LIN {X 0,Y 517.137,Z 472.821,A -85,B 0,C 180,E1 -4939.23,E2 -4939.23} C_VEL
LIN {X 0,Y 516.862,Z 480.781,A -85,B 0,C 180,E1 -4940.412,E2 -4940.412} C_VEL
LIN {X 0,Y 516.641,Z 488.412,A -85,B 0,C 180,E1 -4941.788,E2 -4941.788} C_VEL
LIN {X 0,Y 516.456,Z 493.749,A -85,B 0,C 180,E1 -4942.965,E2 -4942.965} C_VEL
LIN {X 0,Y 516.387,Z 499.361,A -85,B 0,C 180,E1 -4944.533,E2 -4944.533} C_VEL
LIN {X 0,Y 516.343,Z 503.442,A -85,B 0,C 180,E1 -4946.098,E2 -4946.098} C_VEL
LIN {X 0,Y 516.26,Z 506.121,A -85,B 0,C 180,E1 -4947.659,E2 -4947.659} C_VEL
LIN {X 0,Y 516.156,Z 507.471,A -85,B 0,C 180,E1 -4949.22,E2 -4949.22} C_VEL
LIN {X 0,Y 516.157,Z 507.515,A -85,B 0,C 180,E1 -4950.78,E2 -4950.78} C_VEL
LIN {X 0,Y 516.26,Z 506.249,A -85,B 0,C 180,E1 -4952.341,E2 -4952.341} C_VEL
LIN {X 0,Y 516.343,Z 503.644,A -85,B 0,C 180,E1 -4953.902,E2 -4953.902} C_VEL
LIN {X 0,Y 516.381,Z 499.634,A -85,B 0,C 180,E1 -4955.467,E2 -4955.467} C_VEL
LIN {X 0,Y 516.456,Z 494.108,A -85,B 0,C 180,E1 -4957.035,E2 -4957.035} C_VEL
LIN {X 0,Y 516.597,Z 488.866,A -85,B 0,C 180,E1 -4958.213,E2 -4958.213} C_VEL
LIN {X 0,Y 516.842,Z 481.33,A -85,B 0,C 180,E1 -4959.589,E2 -4959.589} C_VEL
LIN {X 0,Y 517.102,Z 473.48,A -85,B 0,C 180,E1 -4960.771,E2 -4960.771} C_VEL
LIN {X 0,Y 517.53,Z 463.302,A -85,B 0,C 180,E1 -4962.032,E2 -4962.032} C_VEL
LIN {X 0,Y 517.893,Z 452.448,A -85,B 0,C 180,E1 -4963.139,E2 -4963.139} C_VEL
LIN {X 0,Y 518.34,Z 440.597,A -85,B 0,C 180,E1 -4964.126,E2 -4964.126} C_VEL
LIN {X 0,Y 518.79,Z 428.907,A -85,B 0,C 180,E1 -4964.916,E2 -4964.916} C_VEL
LIN {X 0,Y 519.149,Z 416.098,A -85,B 0,C 180,E1 -4965.608,E2 -4965.608} C_VEL
LIN {X 0,Y 519.522,Z 402.223,A -85,B 0,C 180,E1 -4966.176,E2 -4966.176} C_VEL
LIN {X 0,Y 519.479,Z 390.943,A -85,B 0,C 180,E1 -4966.522,E2 -4966.522} C_VEL
LIN {X 0,Y 516.431,Z 377.936,A -85,B 0,C 180,E1 -4966.911,E2 -4966.911} C_VEL
LIN {X 0,Y 516.522,Z 371.712,A -85,B 0,C 180,E1 -4970.142,E2 -4970.142} C_VEL
LIN {X 0,Y 516.595,Z 365.792,A -85,B 0,C 180,E1 -4973.237,E2 -4973.237} C_VEL
LIN {X 0,Y 516.693,Z 360.394,A -85,B 0,C 180,E1 -4976.139,E2 -4976.139} C_VEL
LIN {X 0,Y 516.775,Z 356.239,A -85,B 0,C 180,E1 -4978.424,E2 -4978.424} C_VEL
LIN {X 0,Y 516.89,Z 351.438,A -85,B 0,C 180,E1 -4981.11,E2 -4981.11} C_VEL
LIN {X 0,Y 517.015,Z 346.413,A -85,B 0,C 180,E1 -4983.983,E2 -4983.983} C_VEL
LIN {X 0,Y 517.158,Z 341.688,A -85,B 0,C 180,E1 -4986.723,E2 -4986.723} C_VEL
LIN {X 0,Y 517.069,Z 337.486,A -85,B 0,C 180,E1 -4989.218,E2 -4989.218} C_VEL
LIN {X 0,Y 516.936,Z 336.726,A -85,B 0,C 180,E1 -4989.717,E2 -4989.717} C_VEL
LIN {X 0,Y 516.888,Z 336.727,A -85,B 0,C 180,E1 -4992.831,E2 -4992.831} C_VEL
LIN {X 0,Y 516.928,Z 336.721,A -85,B 0,C 180,E1 -4995.01,E2 -4995.01} C_VEL
LIN {X 0,Y 516.918,Z 336.721,A -85,B 0,C 180,E1 -4998.399,E2 -4998.399} C_VEL
LIN {X 0,Y 516.886,Z 336.725,A -85,B 0,C 180,E1 -5001.284,E2 -5001.284} C_VEL
LIN {X 0,Y 516.876,Z 336.724,A -85,B 0,C 180,E1 -5004.22,E2 -5004.22} C_VEL
LIN {X 0,Y 516.9,Z 336.722,A -85,B 0,C 180,E1 -5007.053,E2 -5007.053} C_VEL
LIN {X 0,Y 516.898,Z 336.726,A -85,B 0,C 180,E1 -5009.796,E2 -5009.796} C_VEL
LIN {X 0,Y 516.932,Z 336.717,A -85,B 0,C 180,E1 -5012.467,E2 -5012.467} C_VEL
LIN {X 0,Y 516.915,Z 336.724,A -85,B 0,C 180,E1 -5015.072,E2 -5015.072} C_VEL
LIN {X 0,Y 516.892,Z 336.725,A -85,B 0,C 180,E1 -5018.462,E2 -5018.462} C_VEL
LIN {X 0,Y 516.906,Z 336.72,A -85,B 0,C 180,E1 -5020.955,E2 -5020.955} C_VEL
LIN {X 0,Y 516.916,Z 336.724,A -85,B 0,C 180,E1 -5023.41,E2 -5023.41} C_VEL
LIN {X 0,Y 516.9,Z 336.72,A -85,B 0,C 180,E1 -5025.834,E2 -5025.834} C_VEL
LIN {X 0,Y 516.972,Z 336.715,A -85,B 0,C 180,E1 -5028.234,E2 -5028.234} C_VEL
LIN {X 0,Y 516.969,Z 336.713,A -85,B 0,C 180,E1 -5031.4,E2 -5031.4} C_VEL
LIN {X 0,Y 517.016,Z 336.708,A -85,B 0,C 180,E1 -5033.757,E2 -5033.757} C_VEL
LIN {X 0,Y 517.087,Z 336.696,A -85,B 0,C 180,E1 -5037.663,E2 -5037.663} C_VEL
LIN {X 0,Y 517.1,Z 336.695,A -85,B 0,C 180,E1 -5040.779,E2 -5040.779} C_VEL
LIN {X 0,Y 517.017,Z 336.708,A -85,B 0,C 180,E1 -5043.117,E2 -5043.117} C_VEL
LIN {X 0,Y 517.009,Z 336.708,A -85,B 0,C 180,E1 -5046.243,E2 -5046.243} C_VEL
LIN {X 0,Y 516.948,Z 336.715,A -85,B 0,C 180,E1 -5049.389,E2 -5049.389} C_VEL
LIN {X 0,Y 516.99,Z 336.714,A -85,B 0,C 180,E1 -5051.824,E2 -5051.824} C_VEL
LIN {X 0,Y 516.951,Z 336.72,A -85,B 0,C 180,E1 -5055.146,E2 -5055.146} C_VEL
LIN {X 0,Y 516.93,Z 336.72,A -85,B 0,C 180,E1 -5058.222,E2 -5058.222} C_VEL
LIN {X 0,Y 516.918,Z 336.722,A -85,B 0,C 180,E1 -5060.701,E2 -5060.701} C_VEL
LIN {X 0,Y 516.917,Z 336.721,A -85,B 0,C 180,E1 -5064.072,E2 -5064.072} C_VEL
LIN {X 0,Y 516.93,Z 336.72,A -85,B 0,C 180,E1 -5066.657,E2 -5066.657} C_VEL
LIN {X 0,Y 516.916,Z 336.718,A -85,B 0,C 180,E1 -5069.523,E2 -5069.523} C_VEL
LIN {X 0,Y 516.9,Z 336.724,A -85,B 0,C 180,E1 -5072.543,E2 -5072.543} C_VEL
LIN {X 0,Y 516.887,Z 336.729,A -85,B 0,C 180,E1 -5075.332,E2 -5075.332} C_VEL
LIN {X 0,Y 516.885,Z 336.724,A -85,B 0,C 180,E1 -5077.943,E2 -5077.943} C_VEL
LIN {X 0,Y 516.887,Z 336.725,A -85,B 0,C 180,E1 -5080.741,E2 -5080.741} C_VEL
LIN {X 0,Y 516.886,Z 336.726,A -85,B 0,C 180,E1 -5082.831,E2 -5082.831} C_VEL
LIN {X 0,Y 516.885,Z 336.726,A -85,B 0,C 180,E1 -5086.097,E2 -5086.097} C_VEL
LIN {X 0,Y 516.92,Z 336.722,A -85,B 0,C 180,E1 -5088.398,E2 -5088.398} C_VEL
LIN {X 0,Y 516.919,Z 336.861,A -85,B 0,C 180,E1 -5091.437,E2 -5091.437} C_VEL
LIN {X 0,Y 518.231,Z 343.552,A -85,B 0,C 180,E1 -5093.848,E2 -5093.848} C_VEL
LIN {X 0,Y 518.639,Z 347.942,A -85,B 0,C 180,E1 -5095.31,E2 -5095.31} C_VEL
LIN {X 0,Y 518.251,Z 357.992,A -85,B 0,C 180,E1 -5098.43,E2 -5098.43} C_VEL
LIN {X 0,Y 517.815,Z 368.768,A -85,B 0,C 180,E1 -5101.638,E2 -5101.638} C_VEL
LIN {X 0,Y 517.515,Z 379.281,A -85,B 0,C 180,E1 -5104.673,E2 -5104.673} C_VEL
LIN {X 0,Y 517.245,Z 389.787,A -85,B 0,C 180,E1 -5107.638,E2 -5107.638} C_VEL
LIN {X 0,Y 517.019,Z 399.95,A -85,B 0,C 180,E1 -5110.437,E2 -5110.437} C_VEL
LIN {X 0,Y 520.612,Z 416.224,A -85,B 0,C 180,E1 -5110.856,E2 -5110.856} C_VEL
LIN {X 0,Y 520.274,Z 431.577,A -85,B 0,C 180,E1 -5111.28,E2 -5111.28} C_VEL
LIN {X 0,Y 519.839,Z 447.124,A -85,B 0,C 180,E1 -5111.883,E2 -5111.883} C_VEL
LIN {X 0,Y 519.381,Z 460.906,A -85,B 0,C 180,E1 -5112.579,E2 -5112.579} C_VEL
LIN {X 0,Y 518.872,Z 475.109,A -85,B 0,C 180,E1 -5113.474,E2 -5113.474} C_VEL
LIN {X 0,Y 518.428,Z 487.049,A -85,B 0,C 180,E1 -5114.389,E2 -5114.389} C_VEL
LIN {X 0,Y 517.9,Z 498.835,A -85,B 0,C 180,E1 -5115.46,E2 -5115.46} C_VEL
LIN {X 0,Y 517.518,Z 509.845,A -85,B 0,C 180,E1 -5116.652,E2 -5116.652} C_VEL
LIN {X 0,Y 517.154,Z 519.174,A -85,B 0,C 180,E1 -5117.84,E2 -5117.84} C_VEL
LIN {X 0,Y 516.913,Z 528.292,A -85,B 0,C 180,E1 -5119.225,E2 -5119.225} C_VEL
LIN {X 0,Y 516.637,Z 535.748,A -85,B 0,C 180,E1 -5120.605,E2 -5120.605} C_VEL
LIN {X 0,Y 516.463,Z 542.699,A -85,B 0,C 180,E1 -5122.179,E2 -5122.179} C_VEL
LIN {X 0,Y 516.36,Z 548.161,A -85,B 0,C 180,E1 -5123.749,E2 -5123.749} C_VEL
LIN {X 0,Y 516.238,Z 552.29,A -85,B 0,C 180,E1 -5125.315,E2 -5125.315} C_VEL
LIN {X 0,Y 516.272,Z 555.183,A -85,B 0,C 180,E1 -5126.878,E2 -5126.878} C_VEL
LIN {X 0,Y 516.189,Z 556.909,A -85,B 0,C 180,E1 -5128.44,E2 -5128.44} C_VEL
LIN {X 0,Y 516.151,Z 557.5,A -85,B 0,C 180,E1 -5130,E2 -5130} C_VEL
LIN {X 0,Y 516.189,Z 556.906,A -85,B 0,C 180,E1 -5131.56,E2 -5131.56} C_VEL
LIN {X 0,Y 516.272,Z 555.179,A -85,B 0,C 180,E1 -5133.121,E2 -5133.121} C_VEL
LIN {X 0,Y 516.238,Z 552.288,A -85,B 0,C 180,E1 -5134.685,E2 -5134.685} C_VEL
LIN {X 0,Y 516.376,Z 548.165,A -85,B 0,C 180,E1 -5136.251,E2 -5136.251} C_VEL
LIN {X 0,Y 516.463,Z 542.7,A -85,B 0,C 180,E1 -5137.821,E2 -5137.821} C_VEL
LIN {X 0,Y 516.637,Z 535.742,A -85,B 0,C 180,E1 -5139.395,E2 -5139.395} C_VEL
LIN {X 0,Y 516.91,Z 528.289,A -85,B 0,C 180,E1 -5140.775,E2 -5140.775} C_VEL
LIN {X 0,Y 517.137,Z 519.449,A -85,B 0,C 180,E1 -5142.121,E2 -5142.121} C_VEL
LIN {X 0,Y 517.518,Z 509.847,A -85,B 0,C 180,E1 -5143.348,E2 -5143.348} C_VEL
LIN {X 0,Y 517.882,Z 498.84,A -85,B 0,C 180,E1 -5144.54,E2 -5144.54} C_VEL
LIN {X 0,Y 518.403,Z 487.055,A -85,B 0,C 180,E1 -5145.612,E2 -5145.612} C_VEL
LIN {X 0,Y 518.922,Z 473.663,A -85,B 0,C 180,E1 -5146.625,E2 -5146.625} C_VEL
LIN {X 0,Y 519.373,Z 460.888,A -85,B 0,C 180,E1 -5147.421,E2 -5147.421} C_VEL
LIN {X 0,Y 519.858,Z 447.119,A -85,B 0,C 180,E1 -5148.116,E2 -5148.116} C_VEL
LIN {X 0,Y 520.27,Z 432.263,A -85,B 0,C 180,E1 -5148.697,E2 -5148.697} C_VEL
LIN {X 0,Y 520.606,Z 416.99,A -85,B 0,C 180,E1 -5149.127,E2 -5149.127} C_VEL
LIN {X 0,Y 519.173,Z 409.765,A -85,B 0,C 180,E1 -5149.329,E2 -5149.329} C_VEL
LIN {X 0,Y 517.014,Z 399.848,A -85,B 0,C 180,E1 -5149.591,E2 -5149.591} C_VEL
LIN {X 0,Y 517.303,Z 388.214,A -85,B 0,C 180,E1 -5152.799,E2 -5152.799} C_VEL
LIN {X 0,Y 517.574,Z 376.755,A -85,B 0,C 180,E1 -5156.05,E2 -5156.05} C_VEL
LIN {X 0,Y 517.876,Z 367.26,A -85,B 0,C 180,E1 -5158.801,E2 -5158.801} C_VEL
LIN {X 0,Y 518.305,Z 356.796,A -85,B 0,C 180,E1 -5161.926,E2 -5161.926} C_VEL
LIN {X 0,Y 518.669,Z 347.929,A -85,B 0,C 180,E1 -5164.688,E2 -5164.688} C_VEL
LIN {X 0,Y 518.204,Z 343.555,A -85,B 0,C 180,E1 -5166.154,E2 -5166.154} C_VEL
LIN {X 0,Y 516.897,Z 336.728,A -85,B 0,C 180,E1 -5168.615,E2 -5168.615} C_VEL
LIN {X 0,Y 516.917,Z 336.72,A -85,B 0,C 180,E1 -5171.775,E2 -5171.775} C_VEL
LIN {X 0,Y 516.896,Z 336.724,A -85,B 0,C 180,E1 -5175.007,E2 -5175.007} C_VEL
LIN {X 0,Y 516.925,Z 336.715,A -85,B 0,C 180,E1 -5178.398,E2 -5178.398} C_VEL
LIN {X 0,Y 516.909,Z 336.726,A -85,B 0,C 180,E1 -5181.287,E2 -5181.287} C_VEL
LIN {X 0,Y 516.894,Z 336.725,A -85,B 0,C 180,E1 -5184.222,E2 -5184.222} C_VEL
LIN {X 0,Y 516.898,Z 336.723,A -85,B 0,C 180,E1 -5187.053,E2 -5187.053} C_VEL
LIN {X 0,Y 516.895,Z 336.726,A -85,B 0,C 180,E1 -5189.797,E2 -5189.797} C_VEL
LIN {X 0,Y 516.93,Z 336.718,A -85,B 0,C 180,E1 -5192.468,E2 -5192.468} C_VEL
LIN {X 0,Y 516.915,Z 336.721,A -85,B 0,C 180,E1 -5195.072,E2 -5195.072} C_VEL
LIN {X 0,Y 516.874,Z 336.726,A -85,B 0,C 180,E1 -5197.622,E2 -5197.622} C_VEL
LIN {X 0,Y 516.936,Z 336.718,A -85,B 0,C 180,E1 -5200.13,E2 -5200.13} C_VEL
LIN {X 0,Y 516.926,Z 336.718,A -85,B 0,C 180,E1 -5202.596,E2 -5202.596} C_VEL
LIN {X 0,Y 516.947,Z 336.718,A -85,B 0,C 180,E1 -5205.03,E2 -5205.03} C_VEL
LIN {X 0,Y 517.01,Z 336.712,A -85,B 0,C 180,E1 -5208.235,E2 -5208.235} C_VEL
LIN {X 0,Y 516.961,Z 336.717,A -85,B 0,C 180,E1 -5211.4,E2 -5211.4} C_VEL
LIN {X 0,Y 517.015,Z 336.705,A -85,B 0,C 180,E1 -5213.757,E2 -5213.757} C_VEL
LIN {X 0,Y 517.088,Z 336.696,A -85,B 0,C 180,E1 -5217.663,E2 -5217.663} C_VEL
LIN {X 0,Y 517.098,Z 336.693,A -85,B 0,C 180,E1 -5220.779,E2 -5220.779} C_VEL
LIN {X 0,Y 517.017,Z 336.711,A -85,B 0,C 180,E1 -5223.117,E2 -5223.117} C_VEL
LIN {X 0,Y 517.015,Z 336.708,A -85,B 0,C 180,E1 -5226.243,E2 -5226.243} C_VEL
LIN {X 0,Y 516.948,Z 336.715,A -85,B 0,C 180,E1 -5229.389,E2 -5229.389} C_VEL
LIN {X 0,Y 516.989,Z 336.714,A -85,B 0,C 180,E1 -5231.824,E2 -5231.824} C_VEL
LIN {X 0,Y 516.95,Z 336.719,A -85,B 0,C 180,E1 -5235.147,E2 -5235.147} C_VEL
LIN {X 0,Y 516.93,Z 336.72,A -85,B 0,C 180,E1 -5238.222,E2 -5238.222} C_VEL
LIN {X 0,Y 516.917,Z 336.718,A -85,B 0,C 180,E1 -5240.701,E2 -5240.701} C_VEL
LIN {X 0,Y 516.917,Z 336.717,A -85,B 0,C 180,E1 -5244.072,E2 -5244.072} C_VEL
LIN {X 0,Y 516.929,Z 336.722,A -85,B 0,C 180,E1 -5246.658,E2 -5246.658} C_VEL
LIN {X 0,Y 516.916,Z 336.718,A -85,B 0,C 180,E1 -5249.524,E2 -5249.524} C_VEL
LIN {X 0,Y 516.9,Z 336.721,A -85,B 0,C 180,E1 -5252.543,E2 -5252.543} C_VEL
LIN {X 0,Y 516.87,Z 336.729,A -85,B 0,C 180,E1 -5255.33,E2 -5255.33} C_VEL
LIN {X 0,Y 516.884,Z 336.723,A -85,B 0,C 180,E1 -5257.943,E2 -5257.943} C_VEL
LIN {X 0,Y 516.886,Z 336.724,A -85,B 0,C 180,E1 -5260.742,E2 -5260.742} C_VEL
LIN {X 0,Y 516.887,Z 336.723,A -85,B 0,C 180,E1 -5262.831,E2 -5262.831} C_VEL
LIN {X 0,Y 516.927,Z 336.722,A -85,B 0,C 180,E1 -5265.01,E2 -5265.01} C_VEL
LIN {X 0,Y 516.919,Z 336.723,A -85,B 0,C 180,E1 -5268.398,E2 -5268.398} C_VEL
LIN {X 0,Y 516.928,Z 336.723,A -85,B 0,C 180,E1 -5270.301,E2 -5270.301} C_VEL
LIN {X 0,Y 516.613,Z 337.308,A -85,B 0,C 180,E1 -5270.735,E2 -5270.735} C_VEL
LIN {X 0,Y 514.727,Z 338.994,A -85,B 0,C 180,E1 -5271.571,E2 -5271.571} C_VEL
LIN {X 0,Y 511.152,Z 341.674,A -85,B 0,C 180,E1 -5272.806,E2 -5272.806} C_VEL
LIN {X 0,Y 510.164,Z 342.833,A -85,B 0,C 180,E1 -5273.448,E2 -5273.448} C_VEL
LIN {X 0,Y 510.094,Z 343.201,A -85,B 0,C 180,E1 -5273.666,E2 -5273.666} C_VEL
LIN {X 0,Y 509.938,Z 348.134,A -85,B 0,C 180,E1 -5276.545,E2 -5276.545} C_VEL
LIN {X 0,Y 509.824,Z 352.985,A -85,B 0,C 180,E1 -5279.333,E2 -5279.333} C_VEL
LIN {X 0,Y 509.759,Z 357.776,A -85,B 0,C 180,E1 -5282.046,E2 -5282.046} C_VEL
LIN {X 0,Y 509.606,Z 362.537,A -85,B 0,C 180,E1 -5284.689,E2 -5284.689} C_VEL
LIN {X 0,Y 509.536,Z 367.804,A -85,B 0,C 180,E1 -5287.537,E2 -5287.537} C_VEL
LIN {X 0,Y 509.391,Z 373.764,A -85,B 0,C 180,E1 -5290.663,E2 -5290.663} C_VEL
LIN {X 0,Y 509.412,Z 378.216,A -85,B 0,C 180,E1 -5292.926,E2 -5292.926} C_VEL
LIN {X 0,Y 512.717,Z 392.09,A -85,B 0,C 180,E1 -5293.347,E2 -5293.347} C_VEL
LIN {X 0,Y 512.896,Z 396.194,A -85,B 0,C 180,E1 -5293.467,E2 -5293.467} C_VEL
LIN {X 0,Y 512.642,Z 409.242,A -85,B 0,C 180,E1 -5293.93,E2 -5293.93} C_VEL
LIN {X 0,Y 512.206,Z 422.905,A -85,B 0,C 180,E1 -5294.583,E2 -5294.583} C_VEL
LIN {X 0,Y 511.681,Z 435.853,A -85,B 0,C 180,E1 -5295.381,E2 -5295.381} C_VEL
LIN {X 0,Y 511.265,Z 447.552,A -85,B 0,C 180,E1 -5296.283,E2 -5296.283} C_VEL
LIN {X 0,Y 510.771,Z 458.23,A -85,B 0,C 180,E1 -5297.282,E2 -5297.282} C_VEL
LIN {X 0,Y 510.383,Z 468.772,A -85,B 0,C 180,E1 -5298.483,E2 -5298.483} C_VEL
LIN {X 0,Y 509.953,Z 477.477,A -85,B 0,C 180,E1 -5299.679,E2 -5299.679} C_VEL
LIN {X 0,Y 509.687,Z 485.805,A -85,B 0,C 180,E1 -5301.076,E2 -5301.076} C_VEL
LIN {X 0,Y 509.438,Z 492.525,A -85,B 0,C 180,E1 -5302.469,E2 -5302.469} C_VEL
LIN {X 0,Y 509.365,Z 498.532,A -85,B 0,C 180,E1 -5304.06,E2 -5304.06} C_VEL
LIN {X 0,Y 509.192,Z 501.971,A -85,B 0,C 180,E1 -5305.25,E2 -5305.25} C_VEL
LIN {X 0,Y 509.269,Z 503.813,A -85,B 0,C 180,E1 -5306.043,E2 -5306.043} C_VEL
LIN {X 0,Y 509.189,Z 506.475,A -85,B 0,C 180,E1 -5307.627,E2 -5307.627} C_VEL
LIN {X 0,Y 509.07,Z 507.818,A -85,B 0,C 180,E1 -5309.209,E2 -5309.209} C_VEL
LIN {X 0,Y 509.071,Z 507.86,A -85,B 0,C 180,E1 -5310.791,E2 -5310.791} C_VEL
LIN {X 0,Y 509.188,Z 506.602,A -85,B 0,C 180,E1 -5312.373,E2 -5312.373} C_VEL
LIN {X 0,Y 509.269,Z 504.011,A -85,B 0,C 180,E1 -5313.957,E2 -5313.957} C_VEL
LIN {X 0,Y 509.318,Z 500.02,A -85,B 0,C 180,E1 -5315.543,E2 -5315.543} C_VEL
LIN {X 0,Y 509.419,Z 494.516,A -85,B 0,C 180,E1 -5317.133,E2 -5317.133} C_VEL
LIN {X 0,Y 509.578,Z 489.301,A -85,B 0,C 180,E1 -5318.327,E2 -5318.327} C_VEL
LIN {X 0,Y 509.847,Z 481.794,A -85,B 0,C 180,E1 -5319.722,E2 -5319.722} C_VEL
LIN {X 0,Y 510.155,Z 473.976,A -85,B 0,C 180,E1 -5320.919,E2 -5320.919} C_VEL
LIN {X 0,Y 510.595,Z 464.033,A -85,B 0,C 180,E1 -5322.175,E2 -5322.175} C_VEL
LIN {X 0,Y 510.998,Z 453.021,A -85,B 0,C 180,E1 -5323.319,E2 -5323.319} C_VEL
LIN {X 0,Y 511.491,Z 441.213,A -85,B 0,C 180,E1 -5324.319,E2 -5324.319} C_VEL
LIN {X 0,Y 511.978,Z 429.575,A -85,B 0,C 180,E1 -5325.119,E2 -5325.119} C_VEL
LIN {X 0,Y 512.36,Z 416.84,A -85,B 0,C 180,E1 -5325.821,E2 -5325.821} C_VEL
LIN {X 0,Y 512.762,Z 403.636,A -85,B 0,C 180,E1 -5326.376,E2 -5326.376} C_VEL
LIN {X 0,Y 512.838,Z 392.563,A -85,B 0,C 180,E1 -5326.726,E2 -5326.726} C_VEL
LIN {X 0,Y 509.841,Z 380.168,A -85,B 0,C 180,E1 -5327.115,E2 -5327.115} C_VEL
LIN {X 0,Y 509.379,Z 378.113,A -85,B 0,C 180,E1 -5327.179,E2 -5327.179} C_VEL
LIN {X 0,Y 509.466,Z 372.16,A -85,B 0,C 180,E1 -5330.273,E2 -5330.273} C_VEL
LIN {X 0,Y 509.517,Z 367.488,A -85,B 0,C 180,E1 -5332.72,E2 -5332.72} C_VEL
LIN {X 0,Y 509.604,Z 362.713,A -85,B 0,C 180,E1 -5335.311,E2 -5335.311} C_VEL
LIN {X 0,Y 509.709,Z 357.756,A -85,B 0,C 180,E1 -5338.06,E2 -5338.06} C_VEL
LIN {X 0,Y 509.852,Z 352.06,A -85,B 0,C 180,E1 -5341.281,E2 -5341.281} C_VEL
LIN {X 0,Y 509.979,Z 346.663,A -85,B 0,C 180,E1 -5344.404,E2 -5344.404} C_VEL
LIN {X 0,Y 510.118,Z 341.73,A -85,B 0,C 180,E1 -5347.316,E2 -5347.316} C_VEL
LIN {X 0,Y 509.957,Z 337.852,A -85,B 0,C 180,E1 -5349.66,E2 -5349.66} C_VEL
LIN {X 0,Y 509.844,Z 337.608,A -85,B 0,C 180,E1 -5350.382,E2 -5350.382} C_VEL
LIN {X 0,Y 509.829,Z 337.607,A -85,B 0,C 180,E1 -5353.062,E2 -5353.062} C_VEL
LIN {X 0,Y 509.835,Z 337.601,A -85,B 0,C 180,E1 -5355.793,E2 -5355.793} C_VEL
LIN {X 0,Y 509.86,Z 337.598,A -85,B 0,C 180,E1 -5358.575,E2 -5358.575} C_VEL
LIN {X 0,Y 509.856,Z 337.601,A -85,B 0,C 180,E1 -5361.787,E2 -5361.787} C_VEL
LIN {X 0,Y 509.835,Z 337.604,A -85,B 0,C 180,E1 -5364.622,E2 -5364.622} C_VEL
LIN {X 0,Y 509.867,Z 337.597,A -85,B 0,C 180,E1 -5367.481,E2 -5367.481} C_VEL
LIN {X 0,Y 509.864,Z 337.6,A -85,B 0,C 180,E1 -5370.274,E2 -5370.274} C_VEL
LIN {X 0,Y 509.889,Z 337.597,A -85,B 0,C 180,E1 -5372.944,E2 -5372.944} C_VEL
LIN {X 0,Y 509.871,Z 337.597,A -85,B 0,C 180,E1 -5375.574,E2 -5375.574} C_VEL
LIN {X 0,Y 509.856,Z 337.596,A -85,B 0,C 180,E1 -5378.998,E2 -5378.998} C_VEL
LIN {X 0,Y 509.867,Z 337.601,A -85,B 0,C 180,E1 -5381.516,E2 -5381.516} C_VEL
LIN {X 0,Y 509.86,Z 337.598,A -85,B 0,C 180,E1 -5383.997,E2 -5383.997} C_VEL
LIN {X 0,Y 509.867,Z 337.599,A -85,B 0,C 180,E1 -5386.448,E2 -5386.448} C_VEL
LIN {X 0,Y 509.92,Z 337.591,A -85,B 0,C 180,E1 -5388.875,E2 -5388.875} C_VEL
LIN {X 0,Y 509.956,Z 337.588,A -85,B 0,C 180,E1 -5392.078,E2 -5392.078} C_VEL
LIN {X 0,Y 509.988,Z 337.581,A -85,B 0,C 180,E1 -5394.464,E2 -5394.464} C_VEL
LIN {X 0,Y 510.059,Z 337.572,A -85,B 0,C 180,E1 -5397.631,E2 -5397.631} C_VEL
LIN {X 0,Y 510.07,Z 337.571,A -85,B 0,C 180,E1 -5400.789,E2 -5400.789} C_VEL
LIN {X 0,Y 509.959,Z 337.587,A -85,B 0,C 180,E1 -5403.16,E2 -5403.16} C_VEL
LIN {X 0,Y 509.96,Z 337.586,A -85,B 0,C 180,E1 -5406.33,E2 -5406.33} C_VEL
LIN {X 0,Y 509.91,Z 337.596,A -85,B 0,C 180,E1 -5408.72,E2 -5408.72} C_VEL
LIN {X 0,Y 509.958,Z 337.591,A -85,B 0,C 180,E1 -5411.93,E2 -5411.93} C_VEL
LIN {X 0,Y 509.9,Z 337.599,A -85,B 0,C 180,E1 -5415.241,E2 -5415.241} C_VEL
LIN {X 0,Y 509.888,Z 337.596,A -85,B 0,C 180,E1 -5417.998,E2 -5417.998} C_VEL
LIN {X 0,Y 509.856,Z 337.6,A -85,B 0,C 180,E1 -5421.001,E2 -5421.001} C_VEL
LIN {X 0,Y 509.842,Z 337.605,A -85,B 0,C 180,E1 -5423.563,E2 -5423.563} C_VEL
LIN {X 0,Y 509.916,Z 337.592,A -85,B 0,C 180,E1 -5426.378,E2 -5426.378} C_VEL
LIN {X 0,Y 509.881,Z 337.6,A -85,B 0,C 180,E1 -5428.844,E2 -5428.844} C_VEL
LIN {X 0,Y 509.824,Z 337.604,A -85,B 0,C 180,E1 -5431.59,E2 -5431.59} C_VEL
LIN {X 0,Y 509.858,Z 337.6,A -85,B 0,C 180,E1 -5434.413,E2 -5434.413} C_VEL
LIN {X 0,Y 509.823,Z 337.607,A -85,B 0,C 180,E1 -5437.34,E2 -5437.34} C_VEL
LIN {X 0,Y 509.841,Z 337.605,A -85,B 0,C 180,E1 -5440.382,E2 -5440.382} C_VEL
LIN {X 0,Y 509.826,Z 337.605,A -85,B 0,C 180,E1 -5443.062,E2 -5443.062} C_VEL
LIN {X 0,Y 509.826,Z 337.608,A -85,B 0,C 180,E1 -5445.793,E2 -5445.793} C_VEL
LIN {X 0,Y 509.861,Z 337.602,A -85,B 0,C 180,E1 -5448.574,E2 -5448.574} C_VEL
LIN {X 0,Y 509.86,Z 337.702,A -85,B 0,C 180,E1 -5451.094,E2 -5451.094} C_VEL
LIN {X 0,Y 511.3,Z 345.012,A -85,B 0,C 180,E1 -5453.768,E2 -5453.768} C_VEL
LIN {X 0,Y 511.7,Z 350.138,A -85,B 0,C 180,E1 -5455.495,E2 -5455.495} C_VEL
LIN {X 0,Y 511.286,Z 359.73,A -85,B 0,C 180,E1 -5458.51,E2 -5458.51} C_VEL
LIN {X 0,Y 510.829,Z 370.314,A -85,B 0,C 180,E1 -5461.704,E2 -5461.704} C_VEL
LIN {X 0,Y 510.494,Z 380.675,A -85,B 0,C 180,E1 -5464.736,E2 -5464.736} C_VEL
LIN {X 0,Y 510.208,Z 391.227,A -85,B 0,C 180,E1 -5467.757,E2 -5467.757} C_VEL
LIN {X 0,Y 509.998,Z 399.799,A -85,B 0,C 180,E1 -5470.178,E2 -5470.178} C_VEL
LIN {X 0,Y 513.494,Z 415.649,A -85,B 0,C 180,E1 -5470.596,E2 -5470.596} C_VEL
LIN {X 0,Y 513.832,Z 419.248,A -85,B 0,C 180,E1 -5470.692,E2 -5470.692} C_VEL
LIN {X 0,Y 513.386,Z 435.11,A -85,B 0,C 180,E1 -5471.177,E2 -5471.177} C_VEL
LIN {X 0,Y 512.942,Z 449.643,A -85,B 0,C 180,E1 -5471.786,E2 -5471.786} C_VEL
LIN {X 0,Y 512.385,Z 463.703,A -85,B 0,C 180,E1 -5472.54,E2 -5472.54} C_VEL
LIN {X 0,Y 511.869,Z 477.307,A -85,B 0,C 180,E1 -5473.447,E2 -5473.447} C_VEL
LIN {X 0,Y 511.349,Z 490.45,A -85,B 0,C 180,E1 -5474.515,E2 -5474.515} C_VEL
LIN {X 0,Y 510.771,Z 502.22,A -85,B 0,C 180,E1 -5475.66,E2 -5475.66} C_VEL
LIN {X 0,Y 510.39,Z 512.629,A -85,B 0,C 180,E1 -5476.867,E2 -5476.867} C_VEL
LIN {X 0,Y 509.935,Z 522.67,A -85,B 0,C 180,E1 -5478.25,E2 -5478.25} C_VEL
LIN {X 0,Y 509.716,Z 531.261,A -85,B 0,C 180,E1 -5479.674,E2 -5479.674} C_VEL
LIN {X 0,Y 509.484,Z 539.186,A -85,B 0,C 180,E1 -5481.272,E2 -5481.272} C_VEL
LIN {X 0,Y 509.318,Z 545.482,A -85,B 0,C 180,E1 -5482.866,E2 -5482.866} C_VEL
LIN {X 0,Y 509.284,Z 550.35,A -85,B 0,C 180,E1 -5484.457,E2 -5484.457} C_VEL
LIN {X 0,Y 509.2,Z 553.885,A -85,B 0,C 180,E1 -5486.043,E2 -5486.043} C_VEL
LIN {X 0,Y 509.158,Z 556.188,A -85,B 0,C 180,E1 -5487.627,E2 -5487.627} C_VEL
LIN {X 0,Y 509.071,Z 557.347,A -85,B 0,C 180,E1 -5489.209,E2 -5489.209} C_VEL
LIN {X 0,Y 509.071,Z 557.346,A -85,B 0,C 180,E1 -5490.791,E2 -5490.791} C_VEL
LIN {X 0,Y 509.158,Z 556.184,A -85,B 0,C 180,E1 -5492.373,E2 -5492.373} C_VEL
LIN {X 0,Y 509.2,Z 553.88,A -85,B 0,C 180,E1 -5493.957,E2 -5493.957} C_VEL
LIN {X 0,Y 509.285,Z 550.351,A -85,B 0,C 180,E1 -5495.543,E2 -5495.543} C_VEL
LIN {X 0,Y 509.32,Z 545.488,A -85,B 0,C 180,E1 -5497.134,E2 -5497.134} C_VEL
LIN {X 0,Y 509.484,Z 539.185,A -85,B 0,C 180,E1 -5498.728,E2 -5498.728} C_VEL
LIN {X 0,Y 509.716,Z 531.258,A -85,B 0,C 180,E1 -5500.326,E2 -5500.326} C_VEL
LIN {X 0,Y 509.964,Z 522.478,A -85,B 0,C 180,E1 -5501.777,E2 -5501.777} C_VEL
LIN {X 0,Y 510.389,Z 512.631,A -85,B 0,C 180,E1 -5503.132,E2 -5503.132} C_VEL
LIN {X 0,Y 510.757,Z 502.221,A -85,B 0,C 180,E1 -5504.34,E2 -5504.34} C_VEL
LIN {X 0,Y 511.29,Z 490.455,A -85,B 0,C 180,E1 -5505.487,E2 -5505.487} C_VEL
LIN {X 0,Y 511.864,Z 477.314,A -85,B 0,C 180,E1 -5506.553,E2 -5506.553} C_VEL
LIN {X 0,Y 512.408,Z 463.701,A -85,B 0,C 180,E1 -5507.459,E2 -5507.459} C_VEL
LIN {X 0,Y 512.899,Z 449.641,A -85,B 0,C 180,E1 -5508.215,E2 -5508.215} C_VEL
LIN {X 0,Y 513.407,Z 435.094,A -85,B 0,C 180,E1 -5508.824,E2 -5508.824} C_VEL
LIN {X 0,Y 513.806,Z 419.604,A -85,B 0,C 180,E1 -5509.3,E2 -5509.3} C_VEL
LIN {X 0,Y 513.494,Z 415.662,A -85,B 0,C 180,E1 -5509.403,E2 -5509.403} C_VEL
LIN {X 0,Y 510.11,Z 400.69,A -85,B 0,C 180,E1 -5509.804,E2 -5509.804} C_VEL
LIN {X 0,Y 509.99,Z 399.71,A -85,B 0,C 180,E1 -5509.838,E2 -5509.838} C_VEL
LIN {X 0,Y 510.3,Z 388.157,A -85,B 0,C 180,E1 -5513.111,E2 -5513.111} C_VEL
LIN {X 0,Y 510.569,Z 377.68,A -85,B 0,C 180,E1 -5516.135,E2 -5516.135} C_VEL
LIN {X 0,Y 510.941,Z 367.168,A -85,B 0,C 180,E1 -5519.229,E2 -5519.229} C_VEL
LIN {X 0,Y 511.34,Z 358.222,A -85,B 0,C 180,E1 -5521.948,E2 -5521.948} C_VEL
LIN {X 0,Y 511.738,Z 349.158,A -85,B 0,C 180,E1 -5524.816,E2 -5524.816} C_VEL
LIN {X 0,Y 511.064,Z 343.845,A -85,B 0,C 180,E1 -5526.645,E2 -5526.645} C_VEL
LIN {X 0,Y 509.856,Z 337.606,A -85,B 0,C 180,E1 -5528.97,E2 -5528.97} C_VEL
LIN {X 0,Y 509.862,Z 337.599,A -85,B 0,C 180,E1 -5531.898,E2 -5531.898} C_VEL
LIN {X 0,Y 509.84,Z 337.602,A -85,B 0,C 180,E1 -5535.33,E2 -5535.33} C_VEL
LIN {X 0,Y 509.868,Z 337.593,A -85,B 0,C 180,E1 -5538.576,E2 -5538.576} C_VEL
LIN {X 0,Y 509.862,Z 337.601,A -85,B 0,C 180,E1 -5541.663,E2 -5541.663} C_VEL
LIN {X 0,Y 509.85,Z 337.606,A -85,B 0,C 180,E1 -5544.624,E2 -5544.624} C_VEL
LIN {X 0,Y 509.864,Z 337.601,A -85,B 0,C 180,E1 -5547.481,E2 -5547.481} C_VEL
LIN {X 0,Y 509.862,Z 337.599,A -85,B 0,C 180,E1 -5550.274,E2 -5550.274} C_VEL
LIN {X 0,Y 509.887,Z 337.6,A -85,B 0,C 180,E1 -5552.945,E2 -5552.945} C_VEL
LIN {X 0,Y 509.874,Z 337.596,A -85,B 0,C 180,E1 -5555.574,E2 -5555.574} C_VEL
LIN {X 0,Y 509.827,Z 337.605,A -85,B 0,C 180,E1 -5558.149,E2 -5558.149} C_VEL
LIN {X 0,Y 509.867,Z 337.596,A -85,B 0,C 180,E1 -5560.682,E2 -5560.682} C_VEL
LIN {X 0,Y 509.887,Z 337.598,A -85,B 0,C 180,E1 -5563.175,E2 -5563.175} C_VEL
LIN {X 0,Y 509.869,Z 337.596,A -85,B 0,C 180,E1 -5565.634,E2 -5565.634} C_VEL
LIN {X 0,Y 509.927,Z 337.589,A -85,B 0,C 180,E1 -5568.875,E2 -5568.875} C_VEL
LIN {X 0,Y 509.926,Z 337.59,A -85,B 0,C 180,E1 -5572.078,E2 -5572.078} C_VEL
LIN {X 0,Y 509.986,Z 337.582,A -85,B 0,C 180,E1 -5574.464,E2 -5574.464} C_VEL
LIN {X 0,Y 510.059,Z 337.571,A -85,B 0,C 180,E1 -5577.631,E2 -5577.631} C_VEL
LIN {X 0,Y 510.068,Z 337.569,A -85,B 0,C 180,E1 -5580.79,E2 -5580.79} C_VEL
LIN {X 0,Y 509.959,Z 337.591,A -85,B 0,C 180,E1 -5583.16,E2 -5583.16} C_VEL
LIN {X 0,Y 509.983,Z 337.585,A -85,B 0,C 180,E1 -5586.33,E2 -5586.33} C_VEL
LIN {X 0,Y 509.914,Z 337.592,A -85,B 0,C 180,E1 -5588.72,E2 -5588.72} C_VEL
LIN {X 0,Y 509.957,Z 337.588,A -85,B 0,C 180,E1 -5591.931,E2 -5591.931} C_VEL
LIN {X 0,Y 509.899,Z 337.596,A -85,B 0,C 180,E1 -5595.242,E2 -5595.242} C_VEL
LIN {X 0,Y 509.887,Z 337.595,A -85,B 0,C 180,E1 -5597.999,E2 -5597.999} C_VEL
LIN {X 0,Y 509.855,Z 337.597,A -85,B 0,C 180,E1 -5601.002,E2 -5601.002} C_VEL
LIN {X 0,Y 509.875,Z 337.594,A -85,B 0,C 180,E1 -5604.426,E2 -5604.426} C_VEL
LIN {X 0,Y 509.888,Z 337.597,A -85,B 0,C 180,E1 -5607.056,E2 -5607.056} C_VEL
LIN {X 0,Y 509.862,Z 337.598,A -85,B 0,C 180,E1 -5609.751,E2 -5609.751} C_VEL
LIN {X 0,Y 509.877,Z 337.595,A -85,B 0,C 180,E1 -5612.774,E2 -5612.774} C_VEL
LIN {X 0,Y 509.83,Z 337.604,A -85,B 0,C 180,E1 -5615.578,E2 -5615.578} C_VEL
LIN {X 0,Y 509.854,Z 337.602,A -85,B 0,C 180,E1 -5618.338,E2 -5618.338} C_VEL
LIN {X 0,Y 509.859,Z 337.6,A -85,B 0,C 180,E1 -5621.425,E2 -5621.425} C_VEL
LIN {X 0,Y 509.86,Z 337.599,A -85,B 0,C 180,E1 -5624.668,E2 -5624.668} C_VEL
LIN {X 0,Y 509.861,Z 337.601,A -85,B 0,C 180,E1 -5628.103,E2 -5628.103} C_VEL
LIN {X 0,Y 509.9,Z 337.701,A -85,B 0,C 180,E1 -5630.343,E2 -5630.343} C_VEL
LIN {X 0,Y 510.095,Z 341.555,A -85,B 0,C 180,E1 -5632.683,E2 -5632.683} C_VEL
LIN {X 0,Y 510.094,Z 343.201,A -85,B 0,C 180,E1 -5633.666,E2 -5633.666} C_VEL
LIN {X 0,Y 509.45,Z 344.397,A -85,B 0,C 180,E1 -5634.311,E2 -5634.311} C_VEL
LIN {X 0,Y 506.569,Z 346.569,A -85,B 0,C 180,E1 -5635.352,E2 -5635.352} C_VEL
LIN {X 0,Y 504.089,Z 348.346,A -85,B 0,C 180,E1 -5636.19,E2 -5636.19} C_VEL
LIN {X 0,Y 502.985,Z 349.605,A -85,B 0,C 180,E1 -5636.84,E2 -5636.84} C_VEL
LIN {X 0,Y 502.877,Z 349.996,A -85,B 0,C 180,E1 -5637.061,E2 -5637.061} C_VEL
LIN {X 0,Y 502.761,Z 355.185,A -85,B 0,C 180,E1 -5640.076,E2 -5640.076} C_VEL
LIN {X 0,Y 502.681,Z 359.482,A -85,B 0,C 180,E1 -5642.524,E2 -5642.524} C_VEL
LIN {X 0,Y 502.545,Z 364.564,A -85,B 0,C 180,E1 -5645.37,E2 -5645.37} C_VEL
LIN {X 0,Y 502.463,Z 369.048,A -85,B 0,C 180,E1 -5647.812,E2 -5647.812} C_VEL
LIN {X 0,Y 502.339,Z 373.908,A -85,B 0,C 180,E1 -5650.38,E2 -5650.38} C_VEL
LIN {X 0,Y 502.358,Z 378.329,A -85,B 0,C 180,E1 -5652.649,E2 -5652.649} C_VEL
LIN {X 0,Y 505.974,Z 393.158,A -85,B 0,C 180,E1 -5653.118,E2 -5653.118} C_VEL
LIN {X 0,Y 506.134,Z 397.717,A -85,B 0,C 180,E1 -5653.258,E2 -5653.258} C_VEL
LIN {X 0,Y 505.813,Z 411.196,A -85,B 0,C 180,E1 -5653.758,E2 -5653.758} C_VEL
LIN {X 0,Y 505.412,Z 423.631,A -85,B 0,C 180,E1 -5654.37,E2 -5654.37} C_VEL
LIN {X 0,Y 504.863,Z 436.516,A -85,B 0,C 180,E1 -5655.179,E2 -5655.179} C_VEL
LIN {X 0,Y 504.408,Z 448.16,A -85,B 0,C 180,E1 -5656.093,E2 -5656.093} C_VEL
LIN {X 0,Y 503.875,Z 458.794,A -85,B 0,C 180,E1 -5657.105,E2 -5657.105} C_VEL
LIN {X 0,Y 503.444,Z 469.296,A -85,B 0,C 180,E1 -5658.322,E2 -5658.322} C_VEL
LIN {X 0,Y 502.975,Z 477.966,A -85,B 0,C 180,E1 -5659.534,E2 -5659.534} C_VEL
LIN {X 0,Y 502.68,Z 486.261,A -85,B 0,C 180,E1 -5660.951,E2 -5660.951} C_VEL
LIN {X 0,Y 502.418,Z 492.95,A -85,B 0,C 180,E1 -5662.363,E2 -5662.363} C_VEL
LIN {X 0,Y 502.284,Z 497.566,A -85,B 0,C 180,E1 -5663.573,E2 -5663.573} C_VEL
LIN {X 0,Y 502.176,Z 501.307,A -85,B 0,C 180,E1 -5664.781,E2 -5664.781} C_VEL
LIN {X 0,Y 502.198,Z 504.183,A -85,B 0,C 180,E1 -5665.988,E2 -5665.988} C_VEL
LIN {X 0,Y 502.119,Z 506.83,A -85,B 0,C 180,E1 -5667.594,E2 -5667.594} C_VEL
LIN {X 0,Y 501.987,Z 508.164,A -85,B 0,C 180,E1 -5669.198,E2 -5669.198} C_VEL
LIN {X 0,Y 501.988,Z 508.206,A -85,B 0,C 180,E1 -5670.802,E2 -5670.802} C_VEL
LIN {X 0,Y 502.119,Z 506.954,A -85,B 0,C 180,E1 -5672.407,E2 -5672.407} C_VEL
LIN {X 0,Y 502.198,Z 504.379,A -85,B 0,C 180,E1 -5674.013,E2 -5674.013} C_VEL
LIN {X 0,Y 502.258,Z 500.406,A -85,B 0,C 180,E1 -5675.621,E2 -5675.621} C_VEL
LIN {X 0,Y 502.367,Z 494.928,A -85,B 0,C 180,E1 -5677.233,E2 -5677.233} C_VEL
LIN {X 0,Y 502.565,Z 489.736,A -85,B 0,C 180,E1 -5678.444,E2 -5678.444} C_VEL
LIN {X 0,Y 502.852,Z 482.259,A -85,B 0,C 180,E1 -5679.858,E2 -5679.858} C_VEL
LIN {X 0,Y 503.203,Z 474.473,A -85,B 0,C 180,E1 -5681.072,E2 -5681.072} C_VEL
LIN {X 0,Y 503.611,Z 465.494,A -85,B 0,C 180,E1 -5682.239,E2 -5682.239} C_VEL
LIN {X 0,Y 504.1,Z 454.648,A -85,B 0,C 180,E1 -5683.402,E2 -5683.402} C_VEL
LIN {X 0,Y 504.594,Z 443.109,A -85,B 0,C 180,E1 -5684.416,E2 -5684.416} C_VEL
LIN {X 0,Y 505.126,Z 431.818,A -85,B 0,C 180,E1 -5685.225,E2 -5685.225} C_VEL
LIN {X 0,Y 505.485,Z 419.575,A -85,B 0,C 180,E1 -5685.938,E2 -5685.938} C_VEL
LIN {X 0,Y 505.949,Z 405.734,A -85,B 0,C 180,E1 -5686.553,E2 -5686.553} C_VEL
LIN {X 0,Y 506.113,Z 393.977,A -85,B 0,C 180,E1 -5686.944,E2 -5686.944} C_VEL
LIN {X 0,Y 503.36,Z 382.326,A -85,B 0,C 180,E1 -5687.329,E2 -5687.329} C_VEL
LIN {X 0,Y 502.321,Z 378.296,A -85,B 0,C 180,E1 -5687.451,E2 -5687.451} C_VEL
LIN {X 0,Y 502.412,Z 372.472,A -85,B 0,C 180,E1 -5690.47,E2 -5690.47} C_VEL
LIN {X 0,Y 502.467,Z 367.604,A -85,B 0,C 180,E1 -5693.057,E2 -5693.057} C_VEL
LIN {X 0,Y 502.571,Z 362.838,A -85,B 0,C 180,E1 -5695.691,E2 -5695.691} C_VEL
LIN {X 0,Y 502.664,Z 358.061,A -85,B 0,C 180,E1 -5698.384,E2 -5698.384} C_VEL
LIN {X 0,Y 502.799,Z 353.227,A -85,B 0,C 180,E1 -5701.143,E2 -5701.143} C_VEL
LIN {X 0,Y 502.94,Z 348.372,A -85,B 0,C 180,E1 -5703.984,E2 -5703.984} C_VEL
LIN {X 0,Y 503.091,Z 343.436,A -85,B 0,C 180,E1 -5706.92,E2 -5706.92} C_VEL
LIN {X 0,Y 503.055,Z 340.084,A -85,B 0,C 180,E1 -5708.953,E2 -5708.953} C_VEL
LIN {X 0,Y 502.844,Z 338.482,A -85,B 0,C 180,E1 -5710.01,E2 -5710.01} C_VEL
LIN {X 0,Y 502.778,Z 338.485,A -85,B 0,C 180,E1 -5713.231,E2 -5713.231} C_VEL
LIN {X 0,Y 502.794,Z 338.478,A -85,B 0,C 180,E1 -5715.661,E2 -5715.661} C_VEL
LIN {X 0,Y 502.823,Z 338.473,A -85,B 0,C 180,E1 -5719.005,E2 -5719.005} C_VEL
LIN {X 0,Y 502.798,Z 338.478,A -85,B 0,C 180,E1 -5722.046,E2 -5722.046} C_VEL
LIN {X 0,Y 502.804,Z 338.481,A -85,B 0,C 180,E1 -5725.034,E2 -5725.034} C_VEL
LIN {X 0,Y 502.789,Z 338.481,A -85,B 0,C 180,E1 -5727.916,E2 -5727.916} C_VEL
LIN {X 0,Y 502.83,Z 338.474,A -85,B 0,C 180,E1 -5730.712,E2 -5730.712} C_VEL
LIN {X 0,Y 502.868,Z 338.471,A -85,B 0,C 180,E1 -5733.439,E2 -5733.439} C_VEL
LIN {X 0,Y 502.792,Z 338.479,A -85,B 0,C 180,E1 -5736.086,E2 -5736.086} C_VEL
LIN {X 0,Y 502.79,Z 338.478,A -85,B 0,C 180,E1 -5738.689,E2 -5738.689} C_VEL
LIN {X 0,Y 502.832,Z 338.475,A -85,B 0,C 180,E1 -5741.248,E2 -5741.248} C_VEL
LIN {X 0,Y 502.855,Z 338.471,A -85,B 0,C 180,E1 -5744.6,E2 -5744.6} C_VEL
LIN {X 0,Y 502.883,Z 338.468,A -85,B 0,C 180,E1 -5748.039,E2 -5748.039} C_VEL
LIN {X 0,Y 502.874,Z 338.467,A -85,B 0,C 180,E1 -5751.157,E2 -5751.157} C_VEL
LIN {X 0,Y 502.934,Z 338.464,A -85,B 0,C 180,E1 -5753.581,E2 -5753.581} C_VEL
LIN {X 0,Y 502.904,Z 338.47,A -85,B 0,C 180,E1 -5756.795,E2 -5756.795} C_VEL
LIN {X 0,Y 503.04,Z 338.447,A -85,B 0,C 180,E1 -5759.199,E2 -5759.199} C_VEL
LIN {X 0,Y 502.907,Z 338.466,A -85,B 0,C 180,E1 -5761.601,E2 -5761.601} C_VEL
LIN {X 0,Y 502.902,Z 338.467,A -85,B 0,C 180,E1 -5763.204,E2 -5763.204} C_VEL
LIN {X 0,Y 502.913,Z 338.465,A -85,B 0,C 180,E1 -5766.419,E2 -5766.419} C_VEL
LIN {X 0,Y 502.87,Z 338.472,A -85,B 0,C 180,E1 -5768.843,E2 -5768.843} C_VEL
LIN {X 0,Y 502.9,Z 338.47,A -85,B 0,C 180,E1 -5772.1,E2 -5772.1} C_VEL
LIN {X 0,Y 502.854,Z 338.477,A -85,B 0,C 180,E1 -5775.399,E2 -5775.399} C_VEL
LIN {X 0,Y 502.846,Z 338.474,A -85,B 0,C 180,E1 -5778.12,E2 -5778.12} C_VEL
LIN {X 0,Y 502.834,Z 338.478,A -85,B 0,C 180,E1 -5780.536,E2 -5780.536} C_VEL
LIN {X 0,Y 502.803,Z 338.477,A -85,B 0,C 180,E1 -5783.04,E2 -5783.04} C_VEL
LIN {X 0,Y 502.845,Z 338.475,A -85,B 0,C 180,E1 -5785.675,E2 -5785.675} C_VEL
LIN {X 0,Y 502.844,Z 338.474,A -85,B 0,C 180,E1 -5788.372,E2 -5788.372} C_VEL
LIN {X 0,Y 502.797,Z 338.479,A -85,B 0,C 180,E1 -5791.498,E2 -5791.498} C_VEL
LIN {X 0,Y 502.811,Z 338.478,A -85,B 0,C 180,E1 -5794.444,E2 -5794.444} C_VEL
LIN {X 0,Y 502.785,Z 338.485,A -85,B 0,C 180,E1 -5797.178,E2 -5797.178} C_VEL
LIN {X 0,Y 502.791,Z 338.479,A -85,B 0,C 180,E1 -5800.015,E2 -5800.015} C_VEL
LIN {X 0,Y 502.806,Z 338.483,A -85,B 0,C 180,E1 -5802.199,E2 -5802.199} C_VEL
LIN {X 0,Y 502.789,Z 338.483,A -85,B 0,C 180,E1 -5805.47,E2 -5805.47} C_VEL
LIN {X 0,Y 502.833,Z 338.477,A -85,B 0,C 180,E1 -5807.864,E2 -5807.864} C_VEL
LIN {X 0,Y 502.834,Z 338.616,A -85,B 0,C 180,E1 -5810.768,E2 -5810.768} C_VEL
LIN {X 0,Y 504.327,Z 346.191,A -85,B 0,C 180,E1 -5813.589,E2 -5813.589} C_VEL
LIN {X 0,Y 504.804,Z 350.933,A -85,B 0,C 180,E1 -5815.226,E2 -5815.226} C_VEL
LIN {X 0,Y 504.343,Z 360.257,A -85,B 0,C 180,E1 -5818.215,E2 -5818.215} C_VEL
LIN {X 0,Y 503.857,Z 370.921,A -85,B 0,C 180,E1 -5821.492,E2 -5821.492} C_VEL
LIN {X 0,Y 503.505,Z 380.571,A -85,B 0,C 180,E1 -5824.36,E2 -5824.36} C_VEL
LIN {X 0,Y 503.193,Z 391.349,A -85,B 0,C 180,E1 -5827.513,E2 -5827.513} C_VEL
LIN {X 0,Y 502.954,Z 399.565,A -85,B 0,C 180,E1 -5829.906,E2 -5829.906} C_VEL
LIN {X 0,Y 506.604,Z 416.317,A -85,B 0,C 180,E1 -5830.365,E2 -5830.365} C_VEL
LIN {X 0,Y 507.059,Z 419.412,A -85,B 0,C 180,E1 -5830.457,E2 -5830.457} C_VEL
LIN {X 0,Y 506.589,Z 434.07,A -85,B 0,C 180,E1 -5830.908,E2 -5830.908} C_VEL
LIN {X 0,Y 506.143,Z 448.869,A -85,B 0,C 180,E1 -5831.533,E2 -5831.533} C_VEL
LIN {X 0,Y 505.551,Z 463,A -85,B 0,C 180,E1 -5832.296,E2 -5832.296} C_VEL
LIN {X 0,Y 504.976,Z 476.662,A -85,B 0,C 180,E1 -5833.214,E2 -5833.214} C_VEL
LIN {X 0,Y 504.414,Z 489.155,A -85,B 0,C 180,E1 -5834.234,E2 -5834.234} C_VEL
LIN {X 0,Y 503.788,Z 501.667,A -85,B 0,C 180,E1 -5835.457,E2 -5835.457} C_VEL
LIN {X 0,Y 503.369,Z 512.106,A -85,B 0,C 180,E1 -5836.681,E2 -5836.681} C_VEL
LIN {X 0,Y 502.865,Z 521.93,A -85,B 0,C 180,E1 -5838.045,E2 -5838.045} C_VEL
LIN {X 0,Y 502.742,Z 529.671,A -85,B 0,C 180,E1 -5839.325,E2 -5839.325} C_VEL
LIN {X 0,Y 502.449,Z 536.918,A -85,B 0,C 180,E1 -5840.743,E2 -5840.743} C_VEL
LIN {X 0,Y 502.276,Z 543.633,A -85,B 0,C 180,E1 -5842.361,E2 -5842.361} C_VEL
LIN {X 0,Y 502.167,Z 548.358,A -85,B 0,C 180,E1 -5843.784,E2 -5843.784} C_VEL
LIN {X 0,Y 502.081,Z 551.909,A -85,B 0,C 180,E1 -5845.182,E2 -5845.182} C_VEL
LIN {X 0,Y 502.107,Z 554.868,A -85,B 0,C 180,E1 -5846.79,E2 -5846.79} C_VEL
LIN {X 0,Y 502.033,Z 556.626,A -85,B 0,C 180,E1 -5848.396,E2 -5848.396} C_VEL
LIN {X 0,Y 501.977,Z 557.227,A -85,B 0,C 180,E1 -5850,E2 -5850} C_VEL
LIN {X 0,Y 502.033,Z 556.625,A -85,B 0,C 180,E1 -5851.604,E2 -5851.604} C_VEL
LIN {X 0,Y 502.107,Z 554.865,A -85,B 0,C 180,E1 -5853.21,E2 -5853.21} C_VEL
LIN {X 0,Y 502.081,Z 551.911,A -85,B 0,C 180,E1 -5854.818,E2 -5854.818} C_VEL
LIN {X 0,Y 502.233,Z 547.705,A -85,B 0,C 180,E1 -5856.428,E2 -5856.428} C_VEL
LIN {X 0,Y 502.3,Z 542.115,A -85,B 0,C 180,E1 -5858.043,E2 -5858.043} C_VEL
LIN {X 0,Y 502.462,Z 534.997,A -85,B 0,C 180,E1 -5859.663,E2 -5859.663} C_VEL
LIN {X 0,Y 502.797,Z 527.384,A -85,B 0,C 180,E1 -5861.081,E2 -5861.081} C_VEL
LIN {X 0,Y 503.115,Z 518.194,A -85,B 0,C 180,E1 -5862.505,E2 -5862.505} C_VEL
LIN {X 0,Y 503.573,Z 507.115,A -85,B 0,C 180,E1 -5863.931,E2 -5863.931} C_VEL
LIN {X 0,Y 504.086,Z 495.723,A -85,B 0,C 180,E1 -5865.154,E2 -5865.154} C_VEL
LIN {X 0,Y 504.666,Z 483.217,A -85,B 0,C 180,E1 -5866.276,E2 -5866.276} C_VEL
LIN {X 0,Y 505.273,Z 469.402,A -85,B 0,C 180,E1 -5867.296,E2 -5867.296} C_VEL
LIN {X 0,Y 505.822,Z 455.858,A -85,B 0,C 180,E1 -5868.113,E2 -5868.113} C_VEL
LIN {X 0,Y 506.418,Z 441.17,A -85,B 0,C 180,E1 -5868.813,E2 -5868.813} C_VEL
LIN {X 0,Y 506.848,Z 426.364,A -85,B 0,C 180,E1 -5869.349,E2 -5869.349} C_VEL
LIN {X 0,Y 506.846,Z 417.327,A -85,B 0,C 180,E1 -5869.602,E2 -5869.602} C_VEL
LIN {X 0,Y 503.486,Z 402.282,A -85,B 0,C 180,E1 -5870.027,E2 -5870.027} C_VEL
LIN {X 0,Y 502.953,Z 399.509,A -85,B 0,C 180,E1 -5870.11,E2 -5870.11} C_VEL
LIN {X 0,Y 503.301,Z 388.035,A -85,B 0,C 180,E1 -5873.451,E2 -5873.451} C_VEL
LIN {X 0,Y 503.616,Z 377.574,A -85,B 0,C 180,E1 -5876.523,E2 -5876.523} C_VEL
LIN {X 0,Y 504.016,Z 367.077,A -85,B 0,C 180,E1 -5879.671,E2 -5879.671} C_VEL
LIN {X 0,Y 504.407,Z 358.159,A -85,B 0,C 180,E1 -5882.441,E2 -5882.441} C_VEL
LIN {X 0,Y 504.807,Z 350.808,A -85,B 0,C 180,E1 -5884.807,E2 -5884.807} C_VEL
LIN {X 0,Y 504.297,Z 346.182,A -85,B 0,C 180,E1 -5886.41,E2 -5886.41} C_VEL
LIN {X 0,Y 502.807,Z 338.485,A -85,B 0,C 180,E1 -5889.298,E2 -5889.298} C_VEL
LIN {X 0,Y 502.804,Z 338.479,A -85,B 0,C 180,E1 -5892.199,E2 -5892.199} C_VEL
LIN {X 0,Y 502.787,Z 338.481,A -85,B 0,C 180,E1 -5895.47,E2 -5895.47} C_VEL
LIN {X 0,Y 502.829,Z 338.47,A -85,B 0,C 180,E1 -5898.935,E2 -5898.935} C_VEL
LIN {X 0,Y 502.8,Z 338.479,A -85,B 0,C 180,E1 -5902.047,E2 -5902.047} C_VEL
LIN {X 0,Y 502.813,Z 338.48,A -85,B 0,C 180,E1 -5905.035,E2 -5905.035} C_VEL
LIN {X 0,Y 502.786,Z 338.486,A -85,B 0,C 180,E1 -5907.916,E2 -5907.916} C_VEL
LIN {X 0,Y 502.827,Z 338.475,A -85,B 0,C 180,E1 -5910.713,E2 -5910.713} C_VEL
LIN {X 0,Y 502.866,Z 338.471,A -85,B 0,C 180,E1 -5913.44,E2 -5913.44} C_VEL
LIN {X 0,Y 502.796,Z 338.481,A -85,B 0,C 180,E1 -5916.087,E2 -5916.087} C_VEL
LIN {X 0,Y 502.788,Z 338.477,A -85,B 0,C 180,E1 -5918.689,E2 -5918.689} C_VEL
LIN {X 0,Y 502.833,Z 338.477,A -85,B 0,C 180,E1 -5921.249,E2 -5921.249} C_VEL
LIN {X 0,Y 502.826,Z 338.472,A -85,B 0,C 180,E1 -5923.767,E2 -5923.767} C_VEL
LIN {X 0,Y 502.836,Z 338.476,A -85,B 0,C 180,E1 -5926.255,E2 -5926.255} C_VEL
LIN {X 0,Y 502.897,Z 338.466,A -85,B 0,C 180,E1 -5928.717,E2 -5928.717} C_VEL
LIN {X 0,Y 502.885,Z 338.468,A -85,B 0,C 180,E1 -5931.967,E2 -5931.967} C_VEL
LIN {X 0,Y 502.943,Z 338.459,A -85,B 0,C 180,E1 -5934.387,E2 -5934.387} C_VEL
LIN {X 0,Y 503.029,Z 338.447,A -85,B 0,C 180,E1 -5937.598,E2 -5937.598} C_VEL
LIN {X 0,Y 503.033,Z 338.45,A -85,B 0,C 180,E1 -5940,E2 -5940} C_VEL
LIN {X 0,Y 503.028,Z 338.449,A -85,B 0,C 180,E1 -5942.402,E2 -5942.402} C_VEL
LIN {X 0,Y 502.943,Z 338.46,A -85,B 0,C 180,E1 -5945.614,E2 -5945.614} C_VEL
LIN {X 0,Y 502.905,Z 338.465,A -85,B 0,C 180,E1 -5948.033,E2 -5948.033} C_VEL
LIN {X 0,Y 502.898,Z 338.466,A -85,B 0,C 180,E1 -5951.283,E2 -5951.283} C_VEL
LIN {X 0,Y 502.85,Z 338.471,A -85,B 0,C 180,E1 -5954.571,E2 -5954.571} C_VEL
LIN {X 0,Y 502.86,Z 338.47,A -85,B 0,C 180,E1 -5957.907,E2 -5957.907} C_VEL
LIN {X 0,Y 502.834,Z 338.473,A -85,B 0,C 180,E1 -5960.536,E2 -5960.536} C_VEL
LIN {X 0,Y 502.799,Z 338.479,A -85,B 0,C 180,E1 -5963.04,E2 -5963.04} C_VEL
LIN {X 0,Y 502.845,Z 338.472,A -85,B 0,C 180,E1 -5965.675,E2 -5965.675} C_VEL
LIN {X 0,Y 502.844,Z 338.476,A -85,B 0,C 180,E1 -5968.373,E2 -5968.373} C_VEL
LIN {X 0,Y 502.797,Z 338.48,A -85,B 0,C 180,E1 -5971.499,E2 -5971.499} C_VEL
LIN {X 0,Y 502.808,Z 338.478,A -85,B 0,C 180,E1 -5973.994,E2 -5973.994} C_VEL
LIN {X 0,Y 502.781,Z 338.483,A -85,B 0,C 180,E1 -5977.178,E2 -5977.178} C_VEL
LIN {X 0,Y 502.791,Z 338.483,A -85,B 0,C 180,E1 -5980.015,E2 -5980.015} C_VEL
LIN {X 0,Y 502.806,Z 338.48,A -85,B 0,C 180,E1 -5982.199,E2 -5982.199} C_VEL
LIN {X 0,Y 502.805,Z 338.482,A -85,B 0,C 180,E1 -5985.468,E2 -5985.468} C_VEL
LIN {X 0,Y 502.824,Z 338.479,A -85,B 0,C 180,E1 -5988.934,E2 -5988.934} C_VEL
LIN {X 0,Y 502.859,Z 338.647,A -85,B 0,C 180,E1 -5990.236,E2 -5990.236} C_VEL
LIN {X 0,Y 503.073,Z 341.612,A -85,B 0,C 180,E1 -5992.071,E2 -5992.071} C_VEL
LIN {X 0,Y 502.991,Z 346.561,A -85,B 0,C 180,E1 -5995.049,E2 -5995.049} C_VEL
LIN {X 0,Y 502.877,Z 349.996,A -85,B 0,C 180,E1 -5997.061,E2 -5997.061} C_VEL
LIN {X 0,Y 502.156,Z 351.209,A -85,B 0,C 180,E1 -5997.715,E2 -5997.715} C_VEL
LIN {X 0,Y 499.263,Z 353.403,A -85,B 0,C 180,E1 -5998.771,E2 -5998.771} C_VEL
LIN {X 0,Y 496.83,Z 355.175,A -85,B 0,C 180,E1 -5999.622,E2 -5999.622} C_VEL
LIN {X 0,Y 495.766,Z 356.44,A -85,B 0,C 180,E1 -6000.281,E2 -6000.281} C_VEL
LIN {X 0,Y 495.667,Z 356.838,A -85,B 0,C 180,E1 -6000.505,E2 -6000.505} C_VEL
LIN {X 0,Y 495.574,Z 361.716,A -85,B 0,C 180,E1 -6003.309,E2 -6003.309} C_VEL
LIN {X 0,Y 495.468,Z 365.971,A -85,B 0,C 180,E1 -6005.71,E2 -6005.71} C_VEL
LIN {X 0,Y 495.377,Z 370.803,A -85,B 0,C 180,E1 -6008.354,E2 -6008.354} C_VEL
LIN {X 0,Y 495.299,Z 377.584,A -85,B 0,C 180,E1 -6011.933,E2 -6011.933} C_VEL
LIN {X 0,Y 495.326,Z 378.432,A -85,B 0,C 180,E1 -6012.372,E2 -6012.372} C_VEL
LIN {X 0,Y 499.106,Z 393.646,A -85,B 0,C 180,E1 -6012.862,E2 -6012.862} C_VEL
LIN {X 0,Y 499.441,Z 396.933,A -85,B 0,C 180,E1 -6012.968,E2 -6012.968} C_VEL
LIN {X 0,Y 499.125,Z 410.824,A -85,B 0,C 180,E1 -6013.479,E2 -6013.479} C_VEL
LIN {X 0,Y 498.673,Z 422.587,A -85,B 0,C 180,E1 -6014.049,E2 -6014.049} C_VEL
LIN {X 0,Y 498.141,Z 435.772,A -85,B 0,C 180,E1 -6014.87,E2 -6014.87} C_VEL
LIN {X 0,Y 497.583,Z 447.627,A -85,B 0,C 180,E1 -6015.794,E2 -6015.794} C_VEL
LIN {X 0,Y 497.107,Z 457.445,A -85,B 0,C 180,E1 -6016.718,E2 -6016.718} C_VEL
LIN {X 0,Y 496.57,Z 468.227,A -85,B 0,C 180,E1 -6017.95,E2 -6017.95} C_VEL
LIN {X 0,Y 496.116,Z 477.123,A -85,B 0,C 180,E1 -6019.181,E2 -6019.181} C_VEL
LIN {X 0,Y 495.686,Z 485.626,A -85,B 0,C 180,E1 -6020.616,E2 -6020.616} C_VEL
LIN {X 0,Y 495.498,Z 491.606,A -85,B 0,C 180,E1 -6021.846,E2 -6021.846} C_VEL
LIN {X 0,Y 495.252,Z 497.966,A -85,B 0,C 180,E1 -6023.481,E2 -6023.481} C_VEL
LIN {X 0,Y 495.116,Z 501.691,A -85,B 0,C 180,E1 -6024.706,E2 -6024.706} C_VEL
LIN {X 0,Y 495.129,Z 504.552,A -85,B 0,C 180,E1 -6025.93,E2 -6025.93} C_VEL
LIN {X 0,Y 495.052,Z 507.184,A -85,B 0,C 180,E1 -6027.559,E2 -6027.559} C_VEL
LIN {X 0,Y 494.908,Z 508.511,A -85,B 0,C 180,E1 -6029.186,E2 -6029.186} C_VEL
LIN {X 0,Y 494.908,Z 508.551,A -85,B 0,C 180,E1 -6030.814,E2 -6030.814} C_VEL
LIN {X 0,Y 495.052,Z 507.306,A -85,B 0,C 180,E1 -6032.441,E2 -6032.441} C_VEL
LIN {X 0,Y 495.129,Z 504.745,A -85,B 0,C 180,E1 -6034.07,E2 -6034.07} C_VEL
LIN {X 0,Y 495.201,Z 500.792,A -85,B 0,C 180,E1 -6035.702,E2 -6035.702} C_VEL
LIN {X 0,Y 495.318,Z 495.342,A -85,B 0,C 180,E1 -6037.337,E2 -6037.337} C_VEL
LIN {X 0,Y 495.53,Z 490.172,A -85,B 0,C 180,E1 -6038.564,E2 -6038.564} C_VEL
LIN {X 0,Y 495.845,Z 482.728,A -85,B 0,C 180,E1 -6039.999,E2 -6039.999} C_VEL
LIN {X 0,Y 496.256,Z 474.971,A -85,B 0,C 180,E1 -6041.229,E2 -6041.229} C_VEL
LIN {X 0,Y 496.778,Z 464.963,A -85,B 0,C 180,E1 -6042.536,E2 -6042.536} C_VEL
LIN {X 0,Y 497.205,Z 455.237,A -85,B 0,C 180,E1 -6043.592,E2 -6043.592} C_VEL
LIN {X 0,Y 497.761,Z 443.746,A -85,B 0,C 180,E1 -6044.619,E2 -6044.619} C_VEL
LIN {X 0,Y 498.365,Z 430.937,A -85,B 0,C 180,E1 -6045.542,E2 -6045.542} C_VEL
LIN {X 0,Y 498.876,Z 417.33,A -85,B 0,C 180,E1 -6046.313,E2 -6046.313} C_VEL
LIN {X 0,Y 499.283,Z 403.978,A -85,B 0,C 180,E1 -6046.885,E2 -6046.885} C_VEL
LIN {X 0,Y 499.339,Z 395.019,A -85,B 0,C 180,E1 -6047.181,E2 -6047.181} C_VEL
LIN {X 0,Y 496.512,Z 383.182,A -85,B 0,C 180,E1 -6047.587,E2 -6047.587} C_VEL
LIN {X 0,Y 495.277,Z 378.411,A -85,B 0,C 180,E1 -6047.728,E2 -6047.728} C_VEL
LIN {X 0,Y 495.363,Z 372.609,A -85,B 0,C 180,E1 -6050.775,E2 -6050.775} C_VEL
LIN {X 0,Y 495.421,Z 367.742,A -85,B 0,C 180,E1 -6053.404,E2 -6053.404} C_VEL
LIN {X 0,Y 495.522,Z 362.97,A -85,B 0,C 180,E1 -6056.083,E2 -6056.083} C_VEL
LIN {X 0,Y 495.634,Z 358.169,A -85,B 0,C 180,E1 -6058.824,E2 -6058.824} C_VEL
LIN {X 0,Y 495.778,Z 353.162,A -85,B 0,C 180,E1 -6061.729,E2 -6061.729} C_VEL
LIN {X 0,Y 495.928,Z 348.128,A -85,B 0,C 180,E1 -6064.72,E2 -6064.72} C_VEL
LIN {X 0,Y 496.102,Z 343.479,A -85,B 0,C 180,E1 -6067.529,E2 -6067.529} C_VEL
LIN {X 0,Y 495.903,Z 340.112,A -85,B 0,C 180,E1 -6069.624,E2 -6069.624} C_VEL
LIN {X 0,Y 495.791,Z 339.36,A -85,B 0,C 180,E1 -6070.164,E2 -6070.164} C_VEL
LIN {X 0,Y 495.731,Z 339.363,A -85,B 0,C 180,E1 -6072.883,E2 -6072.883} C_VEL
LIN {X 0,Y 495.738,Z 339.358,A -85,B 0,C 180,E1 -6075.999,E2 -6075.999} C_VEL
LIN {X 0,Y 495.771,Z 339.352,A -85,B 0,C 180,E1 -6079.3,E2 -6079.3} C_VEL
LIN {X 0,Y 495.734,Z 339.357,A -85,B 0,C 180,E1 -6082.439,E2 -6082.439} C_VEL
LIN {X 0,Y 495.783,Z 339.352,A -85,B 0,C 180,E1 -6085.457,E2 -6085.457} C_VEL
LIN {X 0,Y 495.761,Z 339.359,A -85,B 0,C 180,E1 -6088.364,E2 -6088.364} C_VEL
LIN {X 0,Y 495.793,Z 339.355,A -85,B 0,C 180,E1 -6091.507,E2 -6091.507} C_VEL
LIN {X 0,Y 495.796,Z 339.349,A -85,B 0,C 180,E1 -6093.932,E2 -6093.932} C_VEL
LIN {X 0,Y 495.766,Z 339.354,A -85,B 0,C 180,E1 -6097.139,E2 -6097.139} C_VEL
LIN {X 0,Y 495.777,Z 339.357,A -85,B 0,C 180,E1 -6100.11,E2 -6100.11} C_VEL
LIN {X 0,Y 495.771,Z 339.352,A -85,B 0,C 180,E1 -6102.681,E2 -6102.681} C_VEL
LIN {X 0,Y 495.796,Z 339.353,A -85,B 0,C 180,E1 -6105.217,E2 -6105.217} C_VEL
LIN {X 0,Y 495.858,Z 339.346,A -85,B 0,C 180,E1 -6108.555,E2 -6108.555} C_VEL
LIN {X 0,Y 495.878,Z 339.343,A -85,B 0,C 180,E1 -6111.852,E2 -6111.852} C_VEL
LIN {X 0,Y 495.902,Z 339.335,A -85,B 0,C 180,E1 -6114.306,E2 -6114.306} C_VEL
LIN {X 0,Y 495.998,Z 339.323,A -85,B 0,C 180,E1 -6117.564,E2 -6117.564} C_VEL
LIN {X 0,Y 495.99,Z 339.325,A -85,B 0,C 180,E1 -6120.812,E2 -6120.812} C_VEL
LIN {X 0,Y 495.999,Z 339.325,A -85,B 0,C 180,E1 -6122.436,E2 -6122.436} C_VEL
LIN {X 0,Y 495.895,Z 339.338,A -85,B 0,C 180,E1 -6125.693,E2 -6125.693} C_VEL
LIN {X 0,Y 495.842,Z 339.344,A -85,B 0,C 180,E1 -6128.148,E2 -6128.148} C_VEL
LIN {X 0,Y 495.879,Z 339.339,A -85,B 0,C 180,E1 -6131.444,E2 -6131.444} C_VEL
LIN {X 0,Y 495.796,Z 339.351,A -85,B 0,C 180,E1 -6134.783,E2 -6134.783} C_VEL
LIN {X 0,Y 495.787,Z 339.354,A -85,B 0,C 180,E1 -6137.318,E2 -6137.318} C_VEL
LIN {X 0,Y 495.776,Z 339.355,A -85,B 0,C 180,E1 -6139.89,E2 -6139.89} C_VEL
LIN {X 0,Y 495.771,Z 339.353,A -85,B 0,C 180,E1 -6142.862,E2 -6142.862} C_VEL
LIN {X 0,Y 495.796,Z 339.35,A -85,B 0,C 180,E1 -6146.067,E2 -6146.067} C_VEL
LIN {X 0,Y 495.777,Z 339.357,A -85,B 0,C 180,E1 -6148.814,E2 -6148.814} C_VEL
LIN {X 0,Y 495.759,Z 339.358,A -85,B 0,C 180,E1 -6151.725,E2 -6151.725} C_VEL
LIN {X 0,Y 495.78,Z 339.353,A -85,B 0,C 180,E1 -6154.695,E2 -6154.695} C_VEL
LIN {X 0,Y 495.735,Z 339.36,A -85,B 0,C 180,E1 -6157.561,E2 -6157.561} C_VEL
LIN {X 0,Y 495.77,Z 339.357,A -85,B 0,C 180,E1 -6160.699,E2 -6160.699} C_VEL
LIN {X 0,Y 495.73,Z 339.362,A -85,B 0,C 180,E1 -6164.001,E2 -6164.001} C_VEL
LIN {X 0,Y 495.76,Z 339.36,A -85,B 0,C 180,E1 -6167.12,E2 -6167.12} C_VEL
LIN {X 0,Y 495.761,Z 339.36,A -85,B 0,C 180,E1 -6169.953,E2 -6169.953} C_VEL
LIN {X 0,Y 495.774,Z 339.498,A -85,B 0,C 180,E1 -6170.419,E2 -6170.419} C_VEL
LIN {X 0,Y 497.162,Z 346.461,A -85,B 0,C 180,E1 -6173.073,E2 -6173.073} C_VEL
LIN {X 0,Y 497.868,Z 351.758,A -85,B 0,C 180,E1 -6174.959,E2 -6174.959} C_VEL
LIN {X 0,Y 497.424,Z 360.951,A -85,B 0,C 180,E1 -6177.965,E2 -6177.965} C_VEL
LIN {X 0,Y 496.911,Z 371.51,A -85,B 0,C 180,E1 -6181.269,E2 -6181.269} C_VEL
LIN {X 0,Y 496.55,Z 380.448,A -85,B 0,C 180,E1 -6183.975,E2 -6183.975} C_VEL
LIN {X 0,Y 496.21,Z 390.639,A -85,B 0,C 180,E1 -6187.016,E2 -6187.016} C_VEL
LIN {X 0,Y 495.925,Z 399.484,A -85,B 0,C 180,E1 -6189.637,E2 -6189.637} C_VEL
LIN {X 0,Y 499.438,Z 415.796,A -85,B 0,C 180,E1 -6190.089,E2 -6190.089} C_VEL
LIN {X 0,Y 500.27,Z 420.477,A -85,B 0,C 180,E1 -6190.242,E2 -6190.242} C_VEL
LIN {X 0,Y 499.785,Z 434.363,A -85,B 0,C 180,E1 -6190.684,E2 -6190.684} C_VEL
LIN {X 0,Y 499.275,Z 449.118,A -85,B 0,C 180,E1 -6191.322,E2 -6191.322} C_VEL
LIN {X 0,Y 498.634,Z 463.917,A -85,B 0,C 180,E1 -6192.148,E2 -6192.148} C_VEL
LIN {X 0,Y 498.016,Z 477.338,A -85,B 0,C 180,E1 -6193.078,E2 -6193.078} C_VEL
LIN {X 0,Y 497.411,Z 490.191,A -85,B 0,C 180,E1 -6194.159,E2 -6194.159} C_VEL
LIN {X 0,Y 496.805,Z 501.102,A -85,B 0,C 180,E1 -6195.248,E2 -6195.248} C_VEL
LIN {X 0,Y 496.357,Z 511.583,A -85,B 0,C 180,E1 -6196.489,E2 -6196.489} C_VEL
LIN {X 0,Y 495.932,Z 520.459,A -85,B 0,C 180,E1 -6197.727,E2 -6197.727} C_VEL
LIN {X 0,Y 495.693,Z 529.217,A -85,B 0,C 180,E1 -6199.172,E2 -6199.172} C_VEL
LIN {X 0,Y 495.361,Z 536.488,A -85,B 0,C 180,E1 -6200.61,E2 -6200.61} C_VEL
LIN {X 0,Y 495.186,Z 543.229,A -85,B 0,C 180,E1 -6202.251,E2 -6202.251} C_VEL
LIN {X 0,Y 495.07,Z 548.305,A -85,B 0,C 180,E1 -6203.815,E2 -6203.815} C_VEL
LIN {X 0,Y 495.006,Z 551.54,A -85,B 0,C 180,E1 -6205.113,E2 -6205.113} C_VEL
LIN {X 0,Y 495.027,Z 554.511,A -85,B 0,C 180,E1 -6206.744,E2 -6206.744} C_VEL
LIN {X 0,Y 494.959,Z 556.279,A -85,B 0,C 180,E1 -6208.373,E2 -6208.373} C_VEL
LIN {X 0,Y 494.895,Z 556.882,A -85,B 0,C 180,E1 -6210,E2 -6210} C_VEL
LIN {X 0,Y 494.959,Z 556.277,A -85,B 0,C 180,E1 -6211.627,E2 -6211.627} C_VEL
LIN {X 0,Y 495.027,Z 554.51,A -85,B 0,C 180,E1 -6213.255,E2 -6213.255} C_VEL
LIN {X 0,Y 495.006,Z 551.544,A -85,B 0,C 180,E1 -6214.887,E2 -6214.887} C_VEL
LIN {X 0,Y 495.161,Z 547.318,A -85,B 0,C 180,E1 -6216.52,E2 -6216.52} C_VEL
LIN {X 0,Y 495.233,Z 541.705,A -85,B 0,C 180,E1 -6218.159,E2 -6218.159} C_VEL
LIN {X 0,Y 495.397,Z 534.559,A -85,B 0,C 180,E1 -6219.802,E2 -6219.802} C_VEL
LIN {X 0,Y 495.733,Z 526.918,A -85,B 0,C 180,E1 -6221.241,E2 -6221.241} C_VEL
LIN {X 0,Y 496.092,Z 517.7,A -85,B 0,C 180,E1 -6222.685,E2 -6222.685} C_VEL
LIN {X 0,Y 496.596,Z 506.574,A -85,B 0,C 180,E1 -6224.13,E2 -6224.13} C_VEL
LIN {X 0,Y 497.113,Z 495.129,A -85,B 0,C 180,E1 -6225.372,E2 -6225.372} C_VEL
LIN {X 0,Y 497.771,Z 482.571,A -85,B 0,C 180,E1 -6226.508,E2 -6226.508} C_VEL
LIN {X 0,Y 498.421,Z 468.692,A -85,B 0,C 180,E1 -6227.542,E2 -6227.542} C_VEL
LIN {X 0,Y 499,Z 455.084,A -85,B 0,C 180,E1 -6228.369,E2 -6228.369} C_VEL
LIN {X 0,Y 499.617,Z 440.713,A -85,B 0,C 180,E1 -6229.062,E2 -6229.062} C_VEL
LIN {X 0,Y 500.079,Z 425.721,A -85,B 0,C 180,E1 -6229.61,E2 -6229.61} C_VEL
LIN {X 0,Y 500.171,Z 418.991,A -85,B 0,C 180,E1 -6229.805,E2 -6229.805} C_VEL
LIN {X 0,Y 496.958,Z 404.323,A -85,B 0,C 180,E1 -6230.243,E2 -6230.243} C_VEL
LIN {X 0,Y 495.921,Z 399.394,A -85,B 0,C 180,E1 -6230.387,E2 -6230.387} C_VEL
LIN {X 0,Y 496.259,Z 389.386,A -85,B 0,C 180,E1 -6233.362,E2 -6233.362} C_VEL
LIN {X 0,Y 496.6,Z 378.954,A -85,B 0,C 180,E1 -6236.474,E2 -6236.474} C_VEL
LIN {X 0,Y 497.047,Z 368.463,A -85,B 0,C 180,E1 -6239.662,E2 -6239.662} C_VEL
LIN {X 0,Y 497.461,Z 359.569,A -85,B 0,C 180,E1 -6242.47,E2 -6242.47} C_VEL
LIN {X 0,Y 497.862,Z 351.73,A -85,B 0,C 180,E1 -6245.04,E2 -6245.04} C_VEL
LIN {X 0,Y 497.398,Z 347.871,A -85,B 0,C 180,E1 -6246.402,E2 -6246.402} C_VEL
LIN {X 0,Y 495.872,Z 339.919,A -85,B 0,C 180,E1 -6249.406,E2 -6249.406} C_VEL
LIN {X 0,Y 495.761,Z 339.363,A -85,B 0,C 180,E1 -6249.638,E2 -6249.638} C_VEL
LIN {X 0,Y 495.739,Z 339.361,A -85,B 0,C 180,E1 -6252.507,E2 -6252.507} C_VEL
LIN {X 0,Y 495.739,Z 339.36,A -85,B 0,C 180,E1 -6255.141,E2 -6255.141} C_VEL
LIN {X 0,Y 495.763,Z 339.352,A -85,B 0,C 180,E1 -6258.22,E2 -6258.22} C_VEL
LIN {X 0,Y 495.781,Z 339.358,A -85,B 0,C 180,E1 -6261.23,E2 -6261.23} C_VEL
LIN {X 0,Y 495.761,Z 339.361,A -85,B 0,C 180,E1 -6264.463,E2 -6264.463} C_VEL
LIN {X 0,Y 495.77,Z 339.356,A -85,B 0,C 180,E1 -6267.406,E2 -6267.406} C_VEL
LIN {X 0,Y 495.769,Z 339.354,A -85,B 0,C 180,E1 -6270.254,E2 -6270.254} C_VEL
LIN {X 0,Y 495.827,Z 339.35,A -85,B 0,C 180,E1 -6273.251,E2 -6273.251} C_VEL
LIN {X 0,Y 495.756,Z 339.355,A -85,B 0,C 180,E1 -6275.725,E2 -6275.725} C_VEL
LIN {X 0,Y 495.748,Z 339.356,A -85,B 0,C 180,E1 -6278.371,E2 -6278.371} C_VEL
LIN {X 0,Y 495.788,Z 339.352,A -85,B 0,C 180,E1 -6280.972,E2 -6280.972} C_VEL
LIN {X 0,Y 495.782,Z 339.351,A -85,B 0,C 180,E1 -6283.53,E2 -6283.53} C_VEL
LIN {X 0,Y 495.799,Z 339.351,A -85,B 0,C 180,E1 -6286.056,E2 -6286.056} C_VEL
LIN {X 0,Y 495.872,Z 339.342,A -85,B 0,C 180,E1 -6288.555,E2 -6288.555} C_VEL
LIN {X 0,Y 495.841,Z 339.346,A -85,B 0,C 180,E1 -6291.852,E2 -6291.852} C_VEL
LIN {X 0,Y 495.9,Z 339.336,A -85,B 0,C 180,E1 -6294.307,E2 -6294.307} C_VEL
LIN {X 0,Y 495.998,Z 339.323,A -85,B 0,C 180,E1 -6297.564,E2 -6297.564} C_VEL
LIN {X 0,Y 496.004,Z 339.325,A -85,B 0,C 180,E1 -6300,E2 -6300} C_VEL
LIN {X 0,Y 495.997,Z 339.325,A -85,B 0,C 180,E1 -6302.436,E2 -6302.436} C_VEL
LIN {X 0,Y 495.901,Z 339.337,A -85,B 0,C 180,E1 -6305.694,E2 -6305.694} C_VEL
LIN {X 0,Y 495.876,Z 339.341,A -85,B 0,C 180,E1 -6308.148,E2 -6308.148} C_VEL
LIN {X 0,Y 495.873,Z 339.342,A -85,B 0,C 180,E1 -6311.445,E2 -6311.445} C_VEL
LIN {X 0,Y 495.795,Z 339.352,A -85,B 0,C 180,E1 -6314.783,E2 -6314.783} C_VEL
LIN {X 0,Y 495.787,Z 339.35,A -85,B 0,C 180,E1 -6317.319,E2 -6317.319} C_VEL
LIN {X 0,Y 495.776,Z 339.356,A -85,B 0,C 180,E1 -6319.89,E2 -6319.89} C_VEL
LIN {X 0,Y 495.766,Z 339.354,A -85,B 0,C 180,E1 -6322.861,E2 -6322.861} C_VEL
LIN {X 0,Y 495.795,Z 339.35,A -85,B 0,C 180,E1 -6326.068,E2 -6326.068} C_VEL
LIN {X 0,Y 495.776,Z 339.353,A -85,B 0,C 180,E1 -6328.815,E2 -6328.815} C_VEL
LIN {X 0,Y 495.76,Z 339.359,A -85,B 0,C 180,E1 -6331.725,E2 -6331.725} C_VEL
LIN {X 0,Y 495.773,Z 339.354,A -85,B 0,C 180,E1 -6334.694,E2 -6334.694} C_VEL
LIN {X 0,Y 495.733,Z 339.358,A -85,B 0,C 180,E1 -6337.562,E2 -6337.562} C_VEL
LIN {X 0,Y 495.77,Z 339.355,A -85,B 0,C 180,E1 -6340.7,E2 -6340.7} C_VEL
LIN {X 0,Y 495.738,Z 339.361,A -85,B 0,C 180,E1 -6344.001,E2 -6344.001} C_VEL
LIN {X 0,Y 495.73,Z 339.364,A -85,B 0,C 180,E1 -6347.117,E2 -6347.117} C_VEL
LIN {X 0,Y 495.816,Z 339.409,A -85,B 0,C 180,E1 -6350.014,E2 -6350.014} C_VEL
LIN {X 0,Y 496.068,Z 343.321,A -85,B 0,C 180,E1 -6352.468,E2 -6352.468} C_VEL
LIN {X 0,Y 495.947,Z 348.283,A -85,B 0,C 180,E1 -6355.47,E2 -6355.47} C_VEL
LIN {X 0,Y 495.779,Z 353.171,A -85,B 0,C 180,E1 -6358.365,E2 -6358.365} C_VEL
LIN {X 0,Y 495.667,Z 356.838,A -85,B 0,C 180,E1 -6360.505,E2 -6360.505} C_VEL
LIN {X 0,Y 494.962,Z 358.08,A -85,B 0,C 180,E1 -6361.168,E2 -6361.168} C_VEL
LIN {X 0,Y 492.07,Z 360.287,A -85,B 0,C 180,E1 -6362.239,E2 -6362.239} C_VEL
LIN {X 0,Y 489.63,Z 362.075,A -85,B 0,C 180,E1 -6363.101,E2 -6363.101} C_VEL
LIN {X 0,Y 488.564,Z 363.362,A -85,B 0,C 180,E1 -6363.77,E2 -6363.77} C_VEL
LIN {X 0,Y 488.467,Z 363.769,A -85,B 0,C 180,E1 -6363.997,E2 -6363.997} C_VEL
LIN {X 0,Y 488.379,Z 367.725,A -85,B 0,C 180,E1 -6366.238,E2 -6366.238} C_VEL
LIN {X 0,Y 488.279,Z 373.345,A -85,B 0,C 180,E1 -6369.321,E2 -6369.321} C_VEL
LIN {X 0,Y 488.237,Z 378.556,A -85,B 0,C 180,E1 -6372.08,E2 -6372.08} C_VEL
LIN {X 0,Y 492.217,Z 394.149,A -85,B 0,C 180,E1 -6372.597,E2 -6372.597} C_VEL
LIN {X 0,Y 492.74,Z 397.327,A -85,B 0,C 180,E1 -6372.71,E2 -6372.71} C_VEL
LIN {X 0,Y 492.427,Z 410.458,A -85,B 0,C 180,E1 -6373.193,E2 -6373.193} C_VEL
LIN {X 0,Y 491.901,Z 423.338,A -85,B 0,C 180,E1 -6373.823,E2 -6373.823} C_VEL
LIN {X 0,Y 491.341,Z 436.451,A -85,B 0,C 180,E1 -6374.656,E2 -6374.656} C_VEL
LIN {X 0,Y 490.726,Z 448.263,A -85,B 0,C 180,E1 -6375.591,E2 -6375.591} C_VEL
LIN {X 0,Y 490.22,Z 458.042,A -85,B 0,C 180,E1 -6376.528,E2 -6376.528} C_VEL
LIN {X 0,Y 489.713,Z 467.181,A -85,B 0,C 180,E1 -6377.569,E2 -6377.569} C_VEL
LIN {X 0,Y 489.255,Z 476.315,A -85,B 0,C 180,E1 -6378.818,E2 -6378.818} C_VEL
LIN {X 0,Y 488.782,Z 485.012,A -85,B 0,C 180,E1 -6380.273,E2 -6380.273} C_VEL
LIN {X 0,Y 488.469,Z 492.048,A -85,B 0,C 180,E1 -6381.728,E2 -6381.728} C_VEL
LIN {X 0,Y 488.202,Z 498.373,A -85,B 0,C 180,E1 -6383.387,E2 -6383.387} C_VEL
LIN {X 0,Y 488.059,Z 502.074,A -85,B 0,C 180,E1 -6384.629,E2 -6384.629} C_VEL
LIN {X 0,Y 488.063,Z 504.921,A -85,B 0,C 180,E1 -6385.871,E2 -6385.871} C_VEL
LIN {X 0,Y 487.987,Z 507.539,A -85,B 0,C 180,E1 -6387.524,E2 -6387.524} C_VEL
LIN {X 0,Y 487.831,Z 508.857,A -85,B 0,C 180,E1 -6389.175,E2 -6389.175} C_VEL
LIN {X 0,Y 487.831,Z 508.896,A -85,B 0,C 180,E1 -6390.826,E2 -6390.826} C_VEL
LIN {X 0,Y 487.987,Z 507.658,A -85,B 0,C 180,E1 -6392.476,E2 -6392.476} C_VEL
LIN {X 0,Y 488.063,Z 505.113,A -85,B 0,C 180,E1 -6394.129,E2 -6394.129} C_VEL
LIN {X 0,Y 488.149,Z 501.184,A -85,B 0,C 180,E1 -6395.784,E2 -6395.784} C_VEL
LIN {X 0,Y 488.295,Z 495.76,A -85,B 0,C 180,E1 -6397.443,E2 -6397.443} C_VEL
LIN {X 0,Y 488.513,Z 490.623,A -85,B 0,C 180,E1 -6398.688,E2 -6398.688} C_VEL
LIN {X 0,Y 488.862,Z 483.217,A -85,B 0,C 180,E1 -6400.143,E2 -6400.143} C_VEL
LIN {X 0,Y 489.315,Z 475.5,A -85,B 0,C 180,E1 -6401.39,E2 -6401.39} C_VEL
LIN {X 0,Y 489.854,Z 465.83,A -85,B 0,C 180,E1 -6402.68,E2 -6402.68} C_VEL
LIN {X 0,Y 490.342,Z 455.841,A -85,B 0,C 180,E1 -6403.785,E2 -6403.785} C_VEL
LIN {X 0,Y 490.941,Z 444.39,A -85,B 0,C 180,E1 -6404.826,E2 -6404.826} C_VEL
LIN {X 0,Y 491.526,Z 433.204,A -85,B 0,C 180,E1 -6405.657,E2 -6405.657} C_VEL
LIN {X 0,Y 491.986,Z 420.088,A -85,B 0,C 180,E1 -6406.441,E2 -6406.441} C_VEL
LIN {X 0,Y 492.52,Z 406.257,A -85,B 0,C 180,E1 -6407.065,E2 -6407.065} C_VEL
LIN {X 0,Y 492.596,Z 396.195,A -85,B 0,C 180,E1 -6407.419,E2 -6407.419} C_VEL
LIN {X 0,Y 489.5,Z 383.517,A -85,B 0,C 180,E1 -6407.867,E2 -6407.867} C_VEL
LIN {X 0,Y 488.22,Z 378.552,A -85,B 0,C 180,E1 -6408.011,E2 -6408.011} C_VEL
LIN {X 0,Y 488.291,Z 372.772,A -85,B 0,C 180,E1 -6411.09,E2 -6411.09} C_VEL
LIN {X 0,Y 488.377,Z 367.889,A -85,B 0,C 180,E1 -6413.762,E2 -6413.762} C_VEL
LIN {X 0,Y 488.527,Z 362.423,A -85,B 0,C 180,E1 -6416.882,E2 -6416.882} C_VEL
LIN {X 0,Y 488.617,Z 358.289,A -85,B 0,C 180,E1 -6419.278,E2 -6419.278} C_VEL
LIN {X 0,Y 488.759,Z 353.419,A -85,B 0,C 180,E1 -6422.143,E2 -6422.143} C_VEL
LIN {X 0,Y 488.915,Z 348.512,A -85,B 0,C 180,E1 -6425.099,E2 -6425.099} C_VEL
LIN {X 0,Y 489.067,Z 344.147,A -85,B 0,C 180,E1 -6427.78,E2 -6427.78} C_VEL
LIN {X 0,Y 488.768,Z 340.294,A -85,B 0,C 180,E1 -6430.231,E2 -6430.231} C_VEL
LIN {X 0,Y 488.692,Z 340.237,A -85,B 0,C 180,E1 -6433.654,E2 -6433.654} C_VEL
LIN {X 0,Y 488.691,Z 340.238,A -85,B 0,C 180,E1 -6436.346,E2 -6436.346} C_VEL
LIN {X 0,Y 488.738,Z 340.231,A -85,B 0,C 180,E1 -6439.677,E2 -6439.677} C_VEL
LIN {X 0,Y 488.684,Z 340.237,A -85,B 0,C 180,E1 -6442.841,E2 -6442.841} C_VEL
LIN {X 0,Y 488.736,Z 340.229,A -85,B 0,C 180,E1 -6445.887,E2 -6445.887} C_VEL
LIN {X 0,Y 488.697,Z 340.235,A -85,B 0,C 180,E1 -6448.82,E2 -6448.82} C_VEL
LIN {X 0,Y 488.75,Z 340.231,A -85,B 0,C 180,E1 -6451.671,E2 -6451.671} C_VEL
LIN {X 0,Y 488.753,Z 340.227,A -85,B 0,C 180,E1 -6454.444,E2 -6454.444} C_VEL
LIN {X 0,Y 488.729,Z 340.231,A -85,B 0,C 180,E1 -6457.153,E2 -6457.153} C_VEL
LIN {X 0,Y 488.731,Z 340.232,A -85,B 0,C 180,E1 -6459.811,E2 -6459.811} C_VEL
LIN {X 0,Y 488.721,Z 340.23,A -85,B 0,C 180,E1 -6462.423,E2 -6462.423} C_VEL
LIN {X 0,Y 488.768,Z 340.228,A -85,B 0,C 180,E1 -6465,E2 -6465} C_VEL
LIN {X 0,Y 488.812,Z 340.222,A -85,B 0,C 180,E1 -6468.388,E2 -6468.388} C_VEL
LIN {X 0,Y 488.821,Z 340.221,A -85,B 0,C 180,E1 -6471.734,E2 -6471.734} C_VEL
LIN {X 0,Y 488.861,Z 340.212,A -85,B 0,C 180,E1 -6474.224,E2 -6474.224} C_VEL
LIN {X 0,Y 488.966,Z 340.199,A -85,B 0,C 180,E1 -6477.529,E2 -6477.529} C_VEL
LIN {X 0,Y 488.941,Z 340.203,A -85,B 0,C 180,E1 -6480.823,E2 -6480.823} C_VEL
LIN {X 0,Y 488.967,Z 340.201,A -85,B 0,C 180,E1 -6482.471,E2 -6482.471} C_VEL
LIN {X 0,Y 488.854,Z 340.215,A -85,B 0,C 180,E1 -6485.776,E2 -6485.776} C_VEL
LIN {X 0,Y 488.791,Z 340.223,A -85,B 0,C 180,E1 -6488.267,E2 -6488.267} C_VEL
LIN {X 0,Y 488.838,Z 340.217,A -85,B 0,C 180,E1 -6491.612,E2 -6491.612} C_VEL
LIN {X 0,Y 488.768,Z 340.229,A -85,B 0,C 180,E1 -6495,E2 -6495} C_VEL
LIN {X 0,Y 488.76,Z 340.232,A -85,B 0,C 180,E1 -6498.442,E2 -6498.442} C_VEL
LIN {X 0,Y 488.712,Z 340.234,A -85,B 0,C 180,E1 -6501.07,E2 -6501.07} C_VEL
LIN {X 0,Y 488.7,Z 340.24,A -85,B 0,C 180,E1 -6503.745,E2 -6503.745} C_VEL
LIN {X 0,Y 488.796,Z 340.227,A -85,B 0,C 180,E1 -6506.943,E2 -6506.943} C_VEL
LIN {X 0,Y 488.714,Z 340.236,A -85,B 0,C 180,E1 -6510.363,E2 -6510.363} C_VEL
LIN {X 0,Y 488.74,Z 340.234,A -85,B 0,C 180,E1 -6513.484,E2 -6513.484} C_VEL
LIN {X 0,Y 488.693,Z 340.237,A -85,B 0,C 180,E1 -6516.355,E2 -6516.355} C_VEL
LIN {X 0,Y 488.704,Z 340.234,A -85,B 0,C 180,E1 -6519.254,E2 -6519.254} C_VEL
LIN {X 0,Y 488.711,Z 340.233,A -85,B 0,C 180,E1 -6521.599,E2 -6521.599} C_VEL
LIN {X 0,Y 488.704,Z 340.233,A -85,B 0,C 180,E1 -6524.802,E2 -6524.802} C_VEL
LIN {X 0,Y 488.699,Z 340.238,A -85,B 0,C 180,E1 -6527.475,E2 -6527.475} C_VEL
LIN {X 0,Y 488.755,Z 340.422,A -85,B 0,C 180,E1 -6530.082,E2 -6530.082} C_VEL
LIN {X 0,Y 490.436,Z 348.935,A -85,B 0,C 180,E1 -6533.368,E2 -6533.368} C_VEL
LIN {X 0,Y 490.915,Z 353.678,A -85,B 0,C 180,E1 -6535.065,E2 -6535.065} C_VEL
LIN {X 0,Y 490.448,Z 362.473,A -85,B 0,C 180,E1 -6537.981,E2 -6537.981} C_VEL
LIN {X 0,Y 489.897,Z 373.214,A -85,B 0,C 180,E1 -6541.39,E2 -6541.39} C_VEL
LIN {X 0,Y 489.47,Z 383.309,A -85,B 0,C 180,E1 -6544.484,E2 -6544.484} C_VEL
LIN {X 0,Y 489.099,Z 393.648,A -85,B 0,C 180,E1 -6547.617,E2 -6547.617} C_VEL
LIN {X 0,Y 488.889,Z 399.368,A -85,B 0,C 180,E1 -6549.345,E2 -6549.345} C_VEL
LIN {X 0,Y 492.69,Z 416.943,A -85,B 0,C 180,E1 -6549.862,E2 -6549.862} C_VEL
LIN {X 0,Y 493.503,Z 421.262,A -85,B 0,C 180,E1 -6550.014,E2 -6550.014} C_VEL
LIN {X 0,Y 492.956,Z 435.696,A -85,B 0,C 180,E1 -6550.497,E2 -6550.497} C_VEL
LIN {X 0,Y 492.392,Z 450.352,A -85,B 0,C 180,E1 -6551.159,E2 -6551.159} C_VEL
LIN {X 0,Y 491.716,Z 464.809,A -85,B 0,C 180,E1 -6551.996,E2 -6551.996} C_VEL
LIN {X 0,Y 491.059,Z 477.988,A -85,B 0,C 180,E1 -6552.938,E2 -6552.938} C_VEL
LIN {X 0,Y 490.427,Z 490.594,A -85,B 0,C 180,E1 -6554.028,E2 -6554.028} C_VEL
LIN {X 0,Y 489.754,Z 502.365,A -85,B 0,C 180,E1 -6555.243,E2 -6555.243} C_VEL
LIN {X 0,Y 489.285,Z 512.638,A -85,B 0,C 180,E1 -6556.502,E2 -6556.502} C_VEL
LIN {X 0,Y 488.773,Z 522.228,A -85,B 0,C 180,E1 -6557.894,E2 -6557.894} C_VEL
LIN {X 0,Y 488.525,Z 531.026,A -85,B 0,C 180,E1 -6559.431,E2 -6559.431} C_VEL
LIN {X 0,Y 488.252,Z 537.912,A -85,B 0,C 180,E1 -6560.889,E2 -6560.889} C_VEL
LIN {X 0,Y 488.069,Z 544.284,A -85,B 0,C 180,E1 -6562.554,E2 -6562.554} C_VEL
LIN {X 0,Y 488,Z 549.212,A -85,B 0,C 180,E1 -6564.214,E2 -6564.214} C_VEL
LIN {X 0,Y 487.899,Z 552.816,A -85,B 0,C 180,E1 -6565.87,E2 -6565.87} C_VEL
LIN {X 0,Y 487.883,Z 555.189,A -85,B 0,C 180,E1 -6567.523,E2 -6567.523} C_VEL
LIN {X 0,Y 487.831,Z 556.381,A -85,B 0,C 180,E1 -6569.174,E2 -6569.174} C_VEL
LIN {X 0,Y 487.831,Z 556.38,A -85,B 0,C 180,E1 -6570.825,E2 -6570.825} C_VEL
LIN {X 0,Y 487.883,Z 555.187,A -85,B 0,C 180,E1 -6572.477,E2 -6572.477} C_VEL
LIN {X 0,Y 487.899,Z 552.814,A -85,B 0,C 180,E1 -6574.13,E2 -6574.13} C_VEL
LIN {X 0,Y 488.01,Z 549.216,A -85,B 0,C 180,E1 -6575.786,E2 -6575.786} C_VEL
LIN {X 0,Y 488.069,Z 544.29,A -85,B 0,C 180,E1 -6577.446,E2 -6577.446} C_VEL
LIN {X 0,Y 488.252,Z 537.91,A -85,B 0,C 180,E1 -6579.11,E2 -6579.11} C_VEL
LIN {X 0,Y 488.606,Z 529.891,A -85,B 0,C 180,E1 -6580.777,E2 -6580.777} C_VEL
LIN {X 0,Y 488.852,Z 521.054,A -85,B 0,C 180,E1 -6582.285,E2 -6582.285} C_VEL
LIN {X 0,Y 489.344,Z 511.03,A -85,B 0,C 180,E1 -6583.708,E2 -6583.708} C_VEL
LIN {X 0,Y 489.858,Z 500.511,A -85,B 0,C 180,E1 -6584.966,E2 -6584.966} C_VEL
LIN {X 0,Y 490.458,Z 489.014,A -85,B 0,C 180,E1 -6586.126,E2 -6586.126} C_VEL
LIN {X 0,Y 491.177,Z 475.306,A -85,B 0,C 180,E1 -6587.272,E2 -6587.272} C_VEL
LIN {X 0,Y 491.836,Z 461.51,A -85,B 0,C 180,E1 -6588.215,E2 -6588.215} C_VEL
LIN {X 0,Y 492.54,Z 447.246,A -85,B 0,C 180,E1 -6588.997,E2 -6588.997} C_VEL
LIN {X 0,Y 493.06,Z 433.479,A -85,B 0,C 180,E1 -6589.591,E2 -6589.591} C_VEL
LIN {X 0,Y 493.351,Z 420.181,A -85,B 0,C 180,E1 -6590.024,E2 -6590.024} C_VEL
LIN {X 0,Y 490.093,Z 404.797,A -85,B 0,C 180,E1 -6590.504,E2 -6590.504} C_VEL
LIN {X 0,Y 488.887,Z 399.365,A -85,B 0,C 180,E1 -6590.655,E2 -6590.655} C_VEL
LIN {X 0,Y 489.269,Z 389.231,A -85,B 0,C 180,E1 -6593.716,E2 -6593.716} C_VEL
LIN {X 0,Y 489.641,Z 379.134,A -85,B 0,C 180,E1 -6596.785,E2 -6596.785} C_VEL
LIN {X 0,Y 490.071,Z 369.842,A -85,B 0,C 180,E1 -6599.654,E2 -6599.654} C_VEL
LIN {X 0,Y 490.53,Z 360.707,A -85,B 0,C 180,E1 -6602.585,E2 -6602.585} C_VEL
LIN {X 0,Y 490.912,Z 353.656,A -85,B 0,C 180,E1 -6604.935,E2 -6604.935} C_VEL
LIN {X 0,Y 490.379,Z 348.942,A -85,B 0,C 180,E1 -6606.623,E2 -6606.623} C_VEL
LIN {X 0,Y 489.1,Z 342.16,A -85,B 0,C 180,E1 -6609.216,E2 -6609.216} C_VEL
LIN {X 0,Y 488.739,Z 340.235,A -85,B 0,C 180,E1 -6610.053,E2 -6610.053} C_VEL
LIN {X 0,Y 488.711,Z 340.235,A -85,B 0,C 180,E1 -6612.827,E2 -6612.827} C_VEL
LIN {X 0,Y 488.696,Z 340.235,A -85,B 0,C 180,E1 -6615.977,E2 -6615.977} C_VEL
LIN {X 0,Y 488.715,Z 340.227,A -85,B 0,C 180,E1 -6618.585,E2 -6618.585} C_VEL
LIN {X 0,Y 488.75,Z 340.232,A -85,B 0,C 180,E1 -6620.941,E2 -6620.941} C_VEL
LIN {X 0,Y 488.688,Z 340.238,A -85,B 0,C 180,E1 -6623.869,E2 -6623.869} C_VEL
LIN {X 0,Y 488.742,Z 340.232,A -85,B 0,C 180,E1 -6626.878,E2 -6626.878} C_VEL
LIN {X 0,Y 488.727,Z 340.235,A -85,B 0,C 180,E1 -6629.781,E2 -6629.781} C_VEL
LIN {X 0,Y 488.795,Z 340.228,A -85,B 0,C 180,E1 -6633.057,E2 -6633.057} C_VEL
LIN {X 0,Y 488.698,Z 340.238,A -85,B 0,C 180,E1 -6636.255,E2 -6636.255} C_VEL
LIN {X 0,Y 488.75,Z 340.226,A -85,B 0,C 180,E1 -6639.176,E2 -6639.176} C_VEL
LIN {X 0,Y 488.763,Z 340.228,A -85,B 0,C 180,E1 -6641.628,E2 -6641.628} C_VEL
LIN {X 0,Y 488.767,Z 340.228,A -85,B 0,C 180,E1 -6645,E2 -6645} C_VEL
LIN {X 0,Y 488.834,Z 340.22,A -85,B 0,C 180,E1 -6648.388,E2 -6648.388} C_VEL
LIN {X 0,Y 488.79,Z 340.226,A -85,B 0,C 180,E1 -6651.733,E2 -6651.733} C_VEL
LIN {X 0,Y 488.86,Z 340.212,A -85,B 0,C 180,E1 -6654.224,E2 -6654.224} C_VEL
LIN {X 0,Y 488.965,Z 340.198,A -85,B 0,C 180,E1 -6657.529,E2 -6657.529} C_VEL
LIN {X 0,Y 488.975,Z 340.201,A -85,B 0,C 180,E1 -6660,E2 -6660} C_VEL
LIN {X 0,Y 488.964,Z 340.201,A -85,B 0,C 180,E1 -6662.471,E2 -6662.471} C_VEL
LIN {X 0,Y 488.86,Z 340.214,A -85,B 0,C 180,E1 -6665.776,E2 -6665.776} C_VEL
LIN {X 0,Y 488.82,Z 340.221,A -85,B 0,C 180,E1 -6668.266,E2 -6668.266} C_VEL
LIN {X 0,Y 488.835,Z 340.219,A -85,B 0,C 180,E1 -6671.612,E2 -6671.612} C_VEL
LIN {X 0,Y 488.767,Z 340.228,A -85,B 0,C 180,E1 -6675,E2 -6675} C_VEL
LIN {X 0,Y 488.76,Z 340.229,A -85,B 0,C 180,E1 -6678.442,E2 -6678.442} C_VEL
LIN {X 0,Y 488.712,Z 340.231,A -85,B 0,C 180,E1 -6681.071,E2 -6681.071} C_VEL
LIN {X 0,Y 488.697,Z 340.234,A -85,B 0,C 180,E1 -6683.745,E2 -6683.745} C_VEL
LIN {X 0,Y 488.796,Z 340.224,A -85,B 0,C 180,E1 -6686.944,E2 -6686.944} C_VEL
LIN {X 0,Y 488.714,Z 340.236,A -85,B 0,C 180,E1 -6690.363,E2 -6690.363} C_VEL
LIN {X 0,Y 488.738,Z 340.234,A -85,B 0,C 180,E1 -6693.484,E2 -6693.484} C_VEL
LIN {X 0,Y 488.686,Z 340.237,A -85,B 0,C 180,E1 -6696.354,E2 -6696.354} C_VEL
LIN {X 0,Y 488.704,Z 340.234,A -85,B 0,C 180,E1 -6699.254,E2 -6699.254} C_VEL
LIN {X 0,Y 488.71,Z 340.236,A -85,B 0,C 180,E1 -6701.6,E2 -6701.6} C_VEL
LIN {X 0,Y 488.716,Z 340.235,A -85,B 0,C 180,E1 -6704.801,E2 -6704.801} C_VEL
LIN {X 0,Y 488.695,Z 340.238,A -85,B 0,C 180,E1 -6707.475,E2 -6707.475} C_VEL
LIN {X 0,Y 488.785,Z 340.433,A -85,B 0,C 180,E1 -6709.951,E2 -6709.951} C_VEL
LIN {X 0,Y 489.038,Z 344.005,A -85,B 0,C 180,E1 -6712.224,E2 -6712.224} C_VEL
LIN {X 0,Y 488.949,Z 348.539,A -85,B 0,C 180,E1 -6715.015,E2 -6715.015} C_VEL
LIN {X 0,Y 488.755,Z 353.574,A -85,B 0,C 180,E1 -6718.037,E2 -6718.037} C_VEL
LIN {X 0,Y 488.621,Z 358.12,A -85,B 0,C 180,E1 -6720.723,E2 -6720.723} C_VEL
LIN {X 0,Y 488.521,Z 362.923,A -85,B 0,C 180,E1 -6723.514,E2 -6723.514} C_VEL
LIN {X 0,Y 488.467,Z 363.769,A -85,B 0,C 180,E1 -6723.997,E2 -6723.997} C_VEL
LIN {X 0,Y 487.763,Z 365.027,A -85,B 0,C 180,E1 -6724.668,E2 -6724.668} C_VEL
LIN {X 0,Y 484.857,Z 367.276,A -85,B 0,C 180,E1 -6725.753,E2 -6725.753} C_VEL
LIN {X 0,Y 482.411,Z 369.101,A -85,B 0,C 180,E1 -6726.626,E2 -6726.626} C_VEL
LIN {X 0,Y 481.355,Z 370.426,A -85,B 0,C 180,E1 -6727.303,E2 -6727.303} C_VEL
LIN {X 0,Y 481.265,Z 370.848,A -85,B 0,C 180,E1 -6727.533,E2 -6727.533} C_VEL
LIN {X 0,Y 481.159,Z 376.056,A -85,B 0,C 180,E1 -6730.37,E2 -6730.37} C_VEL
LIN {X 0,Y 481.17,Z 378.771,A -85,B 0,C 180,E1 -6731.791,E2 -6731.791} C_VEL
LIN {X 0,Y 485.005,Z 393.236,A -85,B 0,C 180,E1 -6732.272,E2 -6732.272} C_VEL
LIN {X 0,Y 486.01,Z 398.255,A -85,B 0,C 180,E1 -6732.464,E2 -6732.464} C_VEL
LIN {X 0,Y 485.667,Z 411.3,A -85,B 0,C 180,E1 -6732.954,E2 -6732.954} C_VEL
LIN {X 0,Y 485.148,Z 424.044,A -85,B 0,C 180,E1 -6733.592,E2 -6733.592} C_VEL
LIN {X 0,Y 484.544,Z 437.118,A -85,B 0,C 180,E1 -6734.435,E2 -6734.435} C_VEL
LIN {X 0,Y 483.894,Z 448.896,A -85,B 0,C 180,E1 -6735.383,E2 -6735.383} C_VEL
LIN {X 0,Y 483.222,Z 460.562,A -85,B 0,C 180,E1 -6736.544,E2 -6736.544} C_VEL
LIN {X 0,Y 482.647,Z 471.017,A -85,B 0,C 180,E1 -6737.821,E2 -6737.821} C_VEL
LIN {X 0,Y 482.073,Z 479.493,A -85,B 0,C 180,E1 -6739.075,E2 -6739.075} C_VEL
LIN {X 0,Y 481.63,Z 487.678,A -85,B 0,C 180,E1 -6740.551,E2 -6740.551} C_VEL
LIN {X 0,Y 481.335,Z 494.263,A -85,B 0,C 180,E1 -6742.027,E2 -6742.027} C_VEL
LIN {X 0,Y 481.161,Z 499.895,A -85,B 0,C 180,E1 -6743.63,E2 -6743.63} C_VEL
LIN {X 0,Y 480.909,Z 503.503,A -85,B 0,C 180,E1 -6744.97,E2 -6744.97} C_VEL
LIN {X 0,Y 480.999,Z 505.301,A -85,B 0,C 180,E1 -6745.811,E2 -6745.811} C_VEL
LIN {X 0,Y 480.924,Z 507.897,A -85,B 0,C 180,E1 -6747.487,E2 -6747.487} C_VEL
LIN {X 0,Y 480.757,Z 509.204,A -85,B 0,C 180,E1 -6749.162,E2 -6749.162} C_VEL
LIN {X 0,Y 480.758,Z 509.242,A -85,B 0,C 180,E1 -6750.838,E2 -6750.838} C_VEL
LIN {X 0,Y 480.924,Z 508.013,A -85,B 0,C 180,E1 -6752.513,E2 -6752.513} C_VEL
LIN {X 0,Y 480.999,Z 505.487,A -85,B 0,C 180,E1 -6754.19,E2 -6754.19} C_VEL
LIN {X 0,Y 481.002,Z 502.684,A -85,B 0,C 180,E1 -6755.45,E2 -6755.45} C_VEL
LIN {X 0,Y 481.159,Z 499.082,A -85,B 0,C 180,E1 -6756.711,E2 -6756.711} C_VEL
LIN {X 0,Y 481.423,Z 492.878,A -85,B 0,C 180,E1 -6758.394,E2 -6758.394} C_VEL
LIN {X 0,Y 481.785,Z 485.962,A -85,B 0,C 180,E1 -6759.87,E2 -6759.87} C_VEL
LIN {X 0,Y 482.185,Z 478.723,A -85,B 0,C 180,E1 -6761.135,E2 -6761.135} C_VEL
LIN {X 0,Y 482.71,Z 470.039,A -85,B 0,C 180,E1 -6762.398,E2 -6762.398} C_VEL
LIN {X 0,Y 483.17,Z 461.37,A -85,B 0,C 180,E1 -6763.458,E2 -6763.458} C_VEL
LIN {X 0,Y 483.823,Z 451.023,A -85,B 0,C 180,E1 -6764.512,E2 -6764.512} C_VEL
LIN {X 0,Y 484.408,Z 439.732,A -85,B 0,C 180,E1 -6765.462,E2 -6765.462} C_VEL
LIN {X 0,Y 485.056,Z 427.304,A -85,B 0,C 180,E1 -6766.304,E2 -6766.304} C_VEL
LIN {X 0,Y 485.491,Z 415.775,A -85,B 0,C 180,E1 -6766.93,E2 -6766.93} C_VEL
LIN {X 0,Y 485.89,Z 401.623,A -85,B 0,C 180,E1 -6767.514,E2 -6767.514} C_VEL
LIN {X 0,Y 485.792,Z 396.651,A -85,B 0,C 180,E1 -6767.687,E2 -6767.687} C_VEL
LIN {X 0,Y 482.256,Z 382.913,A -85,B 0,C 180,E1 -6768.182,E2 -6768.182} C_VEL
LIN {X 0,Y 481.17,Z 378.681,A -85,B 0,C 180,E1 -6768.321,E2 -6768.321} C_VEL
LIN {X 0,Y 481.225,Z 372.94,A -85,B 0,C 180,E1 -6771.415,E2 -6771.415} C_VEL
LIN {X 0,Y 481.351,Z 368.04,A -85,B 0,C 180,E1 -6774.131,E2 -6774.131} C_VEL
LIN {X 0,Y 481.489,Z 362.944,A -85,B 0,C 180,E1 -6777.079,E2 -6777.079} C_VEL
LIN {X 0,Y 481.589,Z 358.414,A -85,B 0,C 180,E1 -6779.748,E2 -6779.748} C_VEL
LIN {X 0,Y 481.762,Z 353.515,A -85,B 0,C 180,E1 -6782.668,E2 -6782.668} C_VEL
LIN {X 0,Y 481.935,Z 348.58,A -85,B 0,C 180,E1 -6785.685,E2 -6785.685} C_VEL
LIN {X 0,Y 482.062,Z 344.75,A -85,B 0,C 180,E1 -6788.069,E2 -6788.069} C_VEL
LIN {X 0,Y 481.715,Z 341.113,A -85,B 0,C 180,E1 -6790.462,E2 -6790.462} C_VEL
LIN {X 0,Y 481.644,Z 341.118,A -85,B 0,C 180,E1 -6793.3,E2 -6793.3} C_VEL
LIN {X 0,Y 481.662,Z 341.11,A -85,B 0,C 180,E1 -6795.641,E2 -6795.641} C_VEL
LIN {X 0,Y 481.661,Z 341.109,A -85,B 0,C 180,E1 -6798.958,E2 -6798.958} C_VEL
LIN {X 0,Y 481.659,Z 341.111,A -85,B 0,C 180,E1 -6801.993,E2 -6801.993} C_VEL
LIN {X 0,Y 481.693,Z 341.108,A -85,B 0,C 180,E1 -6805.318,E2 -6805.318} C_VEL
LIN {X 0,Y 481.651,Z 341.117,A -85,B 0,C 180,E1 -6808.312,E2 -6808.312} C_VEL
LIN {X 0,Y 481.706,Z 341.107,A -85,B 0,C 180,E1 -6811.219,E2 -6811.219} C_VEL
LIN {X 0,Y 481.706,Z 341.103,A -85,B 0,C 180,E1 -6814.043,E2 -6814.043} C_VEL
LIN {X 0,Y 481.68,Z 341.112,A -85,B 0,C 180,E1 -6816.812,E2 -6816.812} C_VEL
LIN {X 0,Y 481.701,Z 341.104,A -85,B 0,C 180,E1 -6819.503,E2 -6819.503} C_VEL
LIN {X 0,Y 481.698,Z 341.106,A -85,B 0,C 180,E1 -6822.158,E2 -6822.158} C_VEL
LIN {X 0,Y 481.749,Z 341.102,A -85,B 0,C 180,E1 -6824.776,E2 -6824.776} C_VEL
LIN {X 0,Y 481.757,Z 341.101,A -85,B 0,C 180,E1 -6828.215,E2 -6828.215} C_VEL
LIN {X 0,Y 481.767,Z 341.099,A -85,B 0,C 180,E1 -6831.612,E2 -6831.612} C_VEL
LIN {X 0,Y 481.822,Z 341.089,A -85,B 0,C 180,E1 -6834.139,E2 -6834.139} C_VEL
LIN {X 0,Y 481.933,Z 341.076,A -85,B 0,C 180,E1 -6837.492,E2 -6837.492} C_VEL
LIN {X 0,Y 481.893,Z 341.081,A -85,B 0,C 180,E1 -6840.835,E2 -6840.835} C_VEL
LIN {X 0,Y 481.933,Z 341.077,A -85,B 0,C 180,E1 -6842.507,E2 -6842.507} C_VEL
LIN {X 0,Y 481.814,Z 341.092,A -85,B 0,C 180,E1 -6845.86,E2 -6845.86} C_VEL
LIN {X 0,Y 481.746,Z 341.102,A -85,B 0,C 180,E1 -6848.388,E2 -6848.388} C_VEL
LIN {X 0,Y 481.801,Z 341.096,A -85,B 0,C 180,E1 -6851.784,E2 -6851.784} C_VEL
LIN {X 0,Y 481.749,Z 341.106,A -85,B 0,C 180,E1 -6855.224,E2 -6855.224} C_VEL
LIN {X 0,Y 481.717,Z 341.11,A -85,B 0,C 180,E1 -6858.721,E2 -6858.721} C_VEL
LIN {X 0,Y 481.652,Z 341.114,A -85,B 0,C 180,E1 -6861.394,E2 -6861.394} C_VEL
LIN {X 0,Y 481.683,Z 341.11,A -85,B 0,C 180,E1 -6864.113,E2 -6864.113} C_VEL
LIN {X 0,Y 481.751,Z 341.104,A -85,B 0,C 180,E1 -6867.139,E2 -6867.139} C_VEL
LIN {X 0,Y 481.683,Z 341.108,A -85,B 0,C 180,E1 -6869.741,E2 -6869.741} C_VEL
LIN {X 0,Y 481.676,Z 341.111,A -85,B 0,C 180,E1 -6872.674,E2 -6872.674} C_VEL
LIN {X 0,Y 481.647,Z 341.118,A -85,B 0,C 180,E1 -6875.709,E2 -6875.709} C_VEL
LIN {X 0,Y 481.674,Z 341.114,A -85,B 0,C 180,E1 -6878.859,E2 -6878.859} C_VEL
LIN {X 0,Y 481.656,Z 341.116,A -85,B 0,C 180,E1 -6881.913,E2 -6881.913} C_VEL
LIN {X 0,Y 481.657,Z 341.111,A -85,B 0,C 180,E1 -6884.458,E2 -6884.458} C_VEL
LIN {X 0,Y 481.68,Z 341.113,A -85,B 0,C 180,E1 -6886.847,E2 -6886.847} C_VEL
LIN {X 0,Y 481.69,Z 341.195,A -85,B 0,C 180,E1 -6889.669,E2 -6889.669} C_VEL
LIN {X 0,Y 483.408,Z 349.871,A -85,B 0,C 180,E1 -6893.093,E2 -6893.093} C_VEL
LIN {X 0,Y 483.98,Z 355.087,A -85,B 0,C 180,E1 -6894.999,E2 -6894.999} C_VEL
LIN {X 0,Y 483.497,Z 363.862,A -85,B 0,C 180,E1 -6897.957,E2 -6897.957} C_VEL
LIN {X 0,Y 482.908,Z 374.209,A -85,B 0,C 180,E1 -6901.297,E2 -6901.297} C_VEL
LIN {X 0,Y 482.432,Z 384.748,A -85,B 0,C 180,E1 -6904.583,E2 -6904.583} C_VEL
LIN {X 0,Y 482.092,Z 393.464,A -85,B 0,C 180,E1 -6907.274,E2 -6907.274} C_VEL
LIN {X 0,Y 481.893,Z 399.24,A -85,B 0,C 180,E1 -6909.055,E2 -6909.055} C_VEL
LIN {X 0,Y 485.849,Z 417.629,A -85,B 0,C 180,E1 -6909.612,E2 -6909.612} C_VEL
LIN {X 0,Y 486.703,Z 422.116,A -85,B 0,C 180,E1 -6909.781,E2 -6909.781} C_VEL
LIN {X 0,Y 486.149,Z 436.731,A -85,B 0,C 180,E1 -6910.294,E2 -6910.294} C_VEL
LIN {X 0,Y 485.509,Z 451.563,A -85,B 0,C 180,E1 -6910.992,E2 -6910.992} C_VEL
LIN {X 0,Y 484.8,Z 465.689,A -85,B 0,C 180,E1 -6911.839,E2 -6911.839} C_VEL
LIN {X 0,Y 484.107,Z 478.635,A -85,B 0,C 180,E1 -6912.795,E2 -6912.795} C_VEL
LIN {X 0,Y 483.39,Z 491.724,A -85,B 0,C 180,E1 -6913.964,E2 -6913.964} C_VEL
LIN {X 0,Y 482.691,Z 503.601,A -85,B 0,C 180,E1 -6915.238,E2 -6915.238} C_VEL
LIN {X 0,Y 482.192,Z 513.61,A -85,B 0,C 180,E1 -6916.514,E2 -6916.514} C_VEL
LIN {X 0,Y 481.658,Z 523.352,A -85,B 0,C 180,E1 -6917.989,E2 -6917.989} C_VEL
LIN {X 0,Y 481.412,Z 531.59,A -85,B 0,C 180,E1 -6919.485,E2 -6919.485} C_VEL
LIN {X 0,Y 481.12,Z 539.205,A -85,B 0,C 180,E1 -6921.177,E2 -6921.177} C_VEL
LIN {X 0,Y 480.986,Z 545.247,A -85,B 0,C 180,E1 -6922.865,E2 -6922.865} C_VEL
LIN {X 0,Y 480.903,Z 548.825,A -85,B 0,C 180,E1 -6924.128,E2 -6924.128} C_VEL
LIN {X 0,Y 480.803,Z 552.451,A -85,B 0,C 180,E1 -6925.809,E2 -6925.809} C_VEL
LIN {X 0,Y 480.799,Z 554.838,A -85,B 0,C 180,E1 -6927.487,E2 -6927.487} C_VEL
LIN {X 0,Y 480.757,Z 556.036,A -85,B 0,C 180,E1 -6929.162,E2 -6929.162} C_VEL
LIN {X 0,Y 480.757,Z 556.036,A -85,B 0,C 180,E1 -6930.838,E2 -6930.838} C_VEL
LIN {X 0,Y 480.799,Z 554.835,A -85,B 0,C 180,E1 -6932.513,E2 -6932.513} C_VEL
LIN {X 0,Y 480.803,Z 552.449,A -85,B 0,C 180,E1 -6934.191,E2 -6934.191} C_VEL
LIN {X 0,Y 480.919,Z 548.831,A -85,B 0,C 180,E1 -6935.871,E2 -6935.871} C_VEL
LIN {X 0,Y 480.993,Z 543.878,A -85,B 0,C 180,E1 -6937.556,E2 -6937.556} C_VEL
LIN {X 0,Y 481.174,Z 537.461,A -85,B 0,C 180,E1 -6939.245,E2 -6939.245} C_VEL
LIN {X 0,Y 481.543,Z 529.408,A -85,B 0,C 180,E1 -6940.937,E2 -6940.937} C_VEL
LIN {X 0,Y 481.844,Z 520.457,A -85,B 0,C 180,E1 -6942.479,E2 -6942.479} C_VEL
LIN {X 0,Y 482.363,Z 510.474,A -85,B 0,C 180,E1 -6943.91,E2 -6943.91} C_VEL
LIN {X 0,Y 482.925,Z 499.916,A -85,B 0,C 180,E1 -6945.186,E2 -6945.186} C_VEL
LIN {X 0,Y 483.613,Z 487.545,A -85,B 0,C 180,E1 -6946.437,E2 -6946.437} C_VEL
LIN {X 0,Y 484.324,Z 474.621,A -85,B 0,C 180,E1 -6947.524,E2 -6947.524} C_VEL
LIN {X 0,Y 485.014,Z 460.769,A -85,B 0,C 180,E1 -6948.48,E2 -6948.48} C_VEL
LIN {X 0,Y 485.773,Z 446.433,A -85,B 0,C 180,E1 -6949.272,E2 -6949.272} C_VEL
LIN {X 0,Y 486.36,Z 431.651,A -85,B 0,C 180,E1 -6949.906,E2 -6949.906} C_VEL
LIN {X 0,Y 486.498,Z 420.862,A -85,B 0,C 180,E1 -6950.266,E2 -6950.266} C_VEL
LIN {X 0,Y 483.289,Z 405.484,A -85,B 0,C 180,E1 -6950.766,E2 -6950.766} C_VEL
LIN {X 0,Y 481.888,Z 399.192,A -85,B 0,C 180,E1 -6950.957,E2 -6950.957} C_VEL
LIN {X 0,Y 482.268,Z 389.06,A -85,B 0,C 180,E1 -6954.082,E2 -6954.082} C_VEL
LIN {X 0,Y 482.717,Z 378.467,A -85,B 0,C 180,E1 -6957.363,E2 -6957.363} C_VEL
LIN {X 0,Y 483.116,Z 369.732,A -85,B 0,C 180,E1 -6960.125,E2 -6960.125} C_VEL
LIN {X 0,Y 483.552,Z 362.317,A -85,B 0,C 180,E1 -6962.544,E2 -6962.544} C_VEL
LIN {X 0,Y 484.001,Z 355.06,A -85,B 0,C 180,E1 -6964.999,E2 -6964.999} C_VEL
LIN {X 0,Y 483.355,Z 349.875,A -85,B 0,C 180,E1 -6966.899,E2 -6966.899} C_VEL
LIN {X 0,Y 481.889,Z 342.178,A -85,B 0,C 180,E1 -6969.92,E2 -6969.92} C_VEL
LIN {X 0,Y 481.674,Z 341.115,A -85,B 0,C 180,E1 -6970.398,E2 -6970.398} C_VEL
LIN {X 0,Y 481.64,Z 341.111,A -85,B 0,C 180,E1 -6973.3,E2 -6973.3} C_VEL
LIN {X 0,Y 481.655,Z 341.113,A -85,B 0,C 180,E1 -6975.642,E2 -6975.642} C_VEL
LIN {X 0,Y 481.67,Z 341.105,A -85,B 0,C 180,E1 -6978.96,E2 -6978.96} C_VEL
LIN {X 0,Y 481.706,Z 341.111,A -85,B 0,C 180,E1 -6981.144,E2 -6981.144} C_VEL
LIN {X 0,Y 481.672,Z 341.116,A -85,B 0,C 180,E1 -6984.795,E2 -6984.795} C_VEL
LIN {X 0,Y 481.675,Z 341.112,A -85,B 0,C 180,E1 -6987.326,E2 -6987.326} C_VEL
LIN {X 0,Y 481.682,Z 341.109,A -85,B 0,C 180,E1 -6990.259,E2 -6990.259} C_VEL
LIN {X 0,Y 481.749,Z 341.105,A -85,B 0,C 180,E1 -6993.112,E2 -6993.112} C_VEL
LIN {X 0,Y 481.682,Z 341.11,A -85,B 0,C 180,E1 -6995.887,E2 -6995.887} C_VEL
LIN {X 0,Y 481.706,Z 341.103,A -85,B 0,C 180,E1 -6999.028,E2 -6999.028} C_VEL
LIN {X 0,Y 481.708,Z 341.104,A -85,B 0,C 180,E1 -7002.159,E2 -7002.159} C_VEL
LIN {X 0,Y 481.747,Z 341.102,A -85,B 0,C 180,E1 -7004.776,E2 -7004.776} C_VEL
LIN {X 0,Y 481.8,Z 341.098,A -85,B 0,C 180,E1 -7008.216,E2 -7008.216} C_VEL
LIN {X 0,Y 481.744,Z 341.105,A -85,B 0,C 180,E1 -7011.612,E2 -7011.612} C_VEL
LIN {X 0,Y 481.821,Z 341.089,A -85,B 0,C 180,E1 -7014.14,E2 -7014.14} C_VEL
LIN {X 0,Y 481.932,Z 341.074,A -85,B 0,C 180,E1 -7017.493,E2 -7017.493} C_VEL
LIN {X 0,Y 481.946,Z 341.076,A -85,B 0,C 180,E1 -7020,E2 -7020} C_VEL
LIN {X 0,Y 481.931,Z 341.077,A -85,B 0,C 180,E1 -7022.508,E2 -7022.508} C_VEL
LIN {X 0,Y 481.821,Z 341.091,A -85,B 0,C 180,E1 -7025.861,E2 -7025.861} C_VEL
LIN {X 0,Y 481.766,Z 341.1,A -85,B 0,C 180,E1 -7028.388,E2 -7028.388} C_VEL
LIN {X 0,Y 481.8,Z 341.096,A -85,B 0,C 180,E1 -7031.784,E2 -7031.784} C_VEL
LIN {X 0,Y 481.748,Z 341.103,A -85,B 0,C 180,E1 -7035.224,E2 -7035.224} C_VEL
LIN {X 0,Y 481.717,Z 341.106,A -85,B 0,C 180,E1 -7038.722,E2 -7038.722} C_VEL
LIN {X 0,Y 481.651,Z 341.112,A -85,B 0,C 180,E1 -7041.395,E2 -7041.395} C_VEL
LIN {X 0,Y 481.682,Z 341.106,A -85,B 0,C 180,E1 -7044.113,E2 -7044.113} C_VEL
LIN {X 0,Y 481.751,Z 341.101,A -85,B 0,C 180,E1 -7047.139,E2 -7047.139} C_VEL
LIN {X 0,Y 481.683,Z 341.108,A -85,B 0,C 180,E1 -7049.741,E2 -7049.741} C_VEL
LIN {X 0,Y 481.676,Z 341.108,A -85,B 0,C 180,E1 -7052.674,E2 -7052.674} C_VEL
LIN {X 0,Y 481.64,Z 341.114,A -85,B 0,C 180,E1 -7055.709,E2 -7055.709} C_VEL
LIN {X 0,Y 481.674,Z 341.113,A -85,B 0,C 180,E1 -7058.859,E2 -7058.859} C_VEL
LIN {X 0,Y 481.656,Z 341.116,A -85,B 0,C 180,E1 -7061.913,E2 -7061.913} C_VEL
LIN {X 0,Y 481.663,Z 341.112,A -85,B 0,C 180,E1 -7064.457,E2 -7064.457} C_VEL
LIN {X 0,Y 481.651,Z 341.115,A -85,B 0,C 180,E1 -7067.839,E2 -7067.839} C_VEL
LIN {X 0,Y 481.721,Z 341.124,A -85,B 0,C 180,E1 -7069.669,E2 -7069.669} C_VEL
LIN {X 0,Y 482.036,Z 344.648,A -85,B 0,C 180,E1 -7071.935,E2 -7071.935} C_VEL
LIN {X 0,Y 481.925,Z 349.143,A -85,B 0,C 180,E1 -7074.752,E2 -7074.752} C_VEL
LIN {X 0,Y 481.743,Z 354.134,A -85,B 0,C 180,E1 -7077.795,E2 -7077.795} C_VEL
LIN {X 0,Y 481.577,Z 359.854,A -85,B 0,C 180,E1 -7081.21,E2 -7081.21} C_VEL
LIN {X 0,Y 481.423,Z 364.661,A -85,B 0,C 180,E1 -7084.027,E2 -7084.027} C_VEL
LIN {X 0,Y 481.316,Z 369.731,A -85,B 0,C 180,E1 -7086.912,E2 -7086.912} C_VEL
LIN {X 0,Y 481.265,Z 370.848,A -85,B 0,C 180,E1 -7087.533,E2 -7087.533} C_VEL
LIN {X 0,Y 480.571,Z 372.158,A -85,B 0,C 180,E1 -7088.213,E2 -7088.213} C_VEL
LIN {X 0,Y 477.649,Z 374.491,A -85,B 0,C 180,E1 -7089.311,E2 -7089.311} C_VEL
LIN {X 0,Y 475.199,Z 376.385,A -85,B 0,C 180,E1 -7090.195,E2 -7090.195} C_VEL
LIN {X 0,Y 474.166,Z 377.76,A -85,B 0,C 180,E1 -7090.881,E2 -7090.881} C_VEL
LIN {X 0,Y 474.093,Z 378.199,A -85,B 0,C 180,E1 -7091.114,E2 -7091.114} C_VEL
LIN {X 0,Y 474.114,Z 378.875,A -85,B 0,C 180,E1 -7091.48,E2 -7091.48} C_VEL
LIN {X 0,Y 478.305,Z 394.63,A -85,B 0,C 180,E1 -7092.027,E2 -7092.027} C_VEL
LIN {X 0,Y 479.244,Z 399.724,A -85,B 0,C 180,E1 -7092.229,E2 -7092.229} C_VEL
LIN {X 0,Y 478.871,Z 413.24,A -85,B 0,C 180,E1 -7092.764,E2 -7092.764} C_VEL
LIN {X 0,Y 478.312,Z 426.462,A -85,B 0,C 180,E1 -7093.46,E2 -7093.46} C_VEL
LIN {X 0,Y 477.664,Z 439.139,A -85,B 0,C 180,E1 -7094.314,E2 -7094.314} C_VEL
LIN {X 0,Y 476.998,Z 450.622,A -85,B 0,C 180,E1 -7095.276,E2 -7095.276} C_VEL
LIN {X 0,Y 476.351,Z 461.104,A -85,B 0,C 180,E1 -7096.346,E2 -7096.346} C_VEL
LIN {X 0,Y 475.816,Z 469.976,A -85,B 0,C 180,E1 -7097.431,E2 -7097.431} C_VEL
LIN {X 0,Y 475.269,Z 478.67,A -85,B 0,C 180,E1 -7098.701,E2 -7098.701} C_VEL
LIN {X 0,Y 474.745,Z 487.068,A -85,B 0,C 180,E1 -7100.198,E2 -7100.198} C_VEL
LIN {X 0,Y 474.443,Z 492.953,A -85,B 0,C 180,E1 -7101.481,E2 -7101.481} C_VEL
LIN {X 0,Y 474.128,Z 499.212,A -85,B 0,C 180,E1 -7103.19,E2 -7103.19} C_VEL
LIN {X 0,Y 473.954,Z 502.865,A -85,B 0,C 180,E1 -7104.469,E2 -7104.469} C_VEL
LIN {X 0,Y 473.918,Z 505.679,A -85,B 0,C 180,E1 -7105.748,E2 -7105.748} C_VEL
LIN {X 0,Y 473.833,Z 508.256,A -85,B 0,C 180,E1 -7107.45,E2 -7107.45} C_VEL
LIN {X 0,Y 473.686,Z 509.55,A -85,B 0,C 180,E1 -7109.15,E2 -7109.15} C_VEL
LIN {X 0,Y 473.686,Z 509.587,A -85,B 0,C 180,E1 -7110.85,E2 -7110.85} C_VEL
LIN {X 0,Y 473.833,Z 508.369,A -85,B 0,C 180,E1 -7112.55,E2 -7112.55} C_VEL
LIN {X 0,Y 473.918,Z 505.863,A -85,B 0,C 180,E1 -7114.252,E2 -7114.252} C_VEL
LIN {X 0,Y 474.051,Z 501.983,A -85,B 0,C 180,E1 -7115.957,E2 -7115.957} C_VEL
LIN {X 0,Y 474.234,Z 496.622,A -85,B 0,C 180,E1 -7117.665,E2 -7117.665} C_VEL
LIN {X 0,Y 474.51,Z 491.54,A -85,B 0,C 180,E1 -7118.947,E2 -7118.947} C_VEL
LIN {X 0,Y 474.925,Z 484.197,A -85,B 0,C 180,E1 -7120.444,E2 -7120.444} C_VEL
LIN {X 0,Y 475.437,Z 476.539,A -85,B 0,C 180,E1 -7121.728,E2 -7121.728} C_VEL
LIN {X 0,Y 475.991,Z 467.63,A -85,B 0,C 180,E1 -7122.969,E2 -7122.969} C_VEL
LIN {X 0,Y 476.614,Z 456.986,A -85,B 0,C 180,E1 -7124.191,E2 -7124.191} C_VEL
LIN {X 0,Y 477.296,Z 445.588,A -85,B 0,C 180,E1 -7125.26,E2 -7125.26} C_VEL
LIN {X 0,Y 477.942,Z 434.478,A -85,B 0,C 180,E1 -7126.114,E2 -7126.114} C_VEL
LIN {X 0,Y 478.493,Z 421.466,A -85,B 0,C 180,E1 -7126.918,E2 -7126.918} C_VEL
LIN {X 0,Y 479.032,Z 407.825,A -85,B 0,C 180,E1 -7127.561,E2 -7127.561} C_VEL
LIN {X 0,Y 479.105,Z 397.929,A -85,B 0,C 180,E1 -7127.93,E2 -7127.93} C_VEL
LIN {X 0,Y 475.36,Z 383.554,A -85,B 0,C 180,E1 -7128.469,E2 -7128.469} C_VEL
LIN {X 0,Y 474.105,Z 378.86,A -85,B 0,C 180,E1 -7128.616,E2 -7128.616} C_VEL
LIN {X 0,Y 474.164,Z 373.118,A -85,B 0,C 180,E1 -7131.75,E2 -7131.75} C_VEL
LIN {X 0,Y 474.301,Z 368.197,A -85,B 0,C 180,E1 -7134.513,E2 -7134.513} C_VEL
LIN {X 0,Y 474.454,Z 363.377,A -85,B 0,C 180,E1 -7137.336,E2 -7137.336} C_VEL
LIN {X 0,Y 474.562,Z 358.53,A -85,B 0,C 180,E1 -7140.234,E2 -7140.234} C_VEL
LIN {X 0,Y 474.756,Z 353.611,A -85,B 0,C 180,E1 -7143.212,E2 -7143.212} C_VEL
LIN {X 0,Y 474.965,Z 348.649,A -85,B 0,C 180,E1 -7146.291,E2 -7146.291} C_VEL
LIN {X 0,Y 475.012,Z 345.303,A -85,B 0,C 180,E1 -7148.419,E2 -7148.419} C_VEL
LIN {X 0,Y 474.658,Z 341.992,A -85,B 0,C 180,E1 -7150.654,E2 -7150.654} C_VEL
LIN {X 0,Y 474.606,Z 341.993,A -85,B 0,C 180,E1 -7153.481,E2 -7153.481} C_VEL
LIN {X 0,Y 474.606,Z 341.992,A -85,B 0,C 180,E1 -7156.519,E2 -7156.519} C_VEL
LIN {X 0,Y 474.621,Z 341.987,A -85,B 0,C 180,E1 -7159.342,E2 -7159.342} C_VEL
LIN {X 0,Y 474.615,Z 341.991,A -85,B 0,C 180,E1 -7161.704,E2 -7161.704} C_VEL
LIN {X 0,Y 474.629,Z 341.991,A -85,B 0,C 180,E1 -7164.726,E2 -7164.726} C_VEL
LIN {X 0,Y 474.641,Z 341.986,A -85,B 0,C 180,E1 -7167.788,E2 -7167.788} C_VEL
LIN {X 0,Y 474.629,Z 341.987,A -85,B 0,C 180,E1 -7170.885,E2 -7170.885} C_VEL
LIN {X 0,Y 474.666,Z 341.982,A -85,B 0,C 180,E1 -7173.629,E2 -7173.629} C_VEL
LIN {X 0,Y 474.641,Z 341.988,A -85,B 0,C 180,E1 -7176.641,E2 -7176.641} C_VEL
LIN {X 0,Y 474.66,Z 341.988,A -85,B 0,C 180,E1 -7180.09,E2 -7180.09} C_VEL
LIN {X 0,Y 474.645,Z 341.984,A -85,B 0,C 180,E1 -7182.774,E2 -7182.774} C_VEL
LIN {X 0,Y 474.654,Z 341.985,A -85,B 0,C 180,E1 -7185.421,E2 -7185.421} C_VEL
LIN {X 0,Y 474.711,Z 341.977,A -85,B 0,C 180,E1 -7188.038,E2 -7188.038} C_VEL
LIN {X 0,Y 474.732,Z 341.975,A -85,B 0,C 180,E1 -7191.486,E2 -7191.486} C_VEL
LIN {X 0,Y 474.785,Z 341.966,A -85,B 0,C 180,E1 -7194.052,E2 -7194.052} C_VEL
LIN {X 0,Y 474.899,Z 341.952,A -85,B 0,C 180,E1 -7197.455,E2 -7197.455} C_VEL
LIN {X 0,Y 474.917,Z 341.955,A -85,B 0,C 180,E1 -7200,E2 -7200} C_VEL
LIN {X 0,Y 474.899,Z 341.953,A -85,B 0,C 180,E1 -7202.544,E2 -7202.544} C_VEL
LIN {X 0,Y 474.777,Z 341.968,A -85,B 0,C 180,E1 -7205.947,E2 -7205.947} C_VEL
LIN {X 0,Y 474.717,Z 341.978,A -85,B 0,C 180,E1 -7208.514,E2 -7208.514} C_VEL
LIN {X 0,Y 474.745,Z 341.978,A -85,B 0,C 180,E1 -7211.961,E2 -7211.961} C_VEL
LIN {X 0,Y 474.686,Z 341.983,A -85,B 0,C 180,E1 -7215.768,E2 -7215.768} C_VEL
LIN {X 0,Y 474.67,Z 341.984,A -85,B 0,C 180,E1 -7219.01,E2 -7219.01} C_VEL
LIN {X 0,Y 474.597,Z 341.996,A -85,B 0,C 180,E1 -7221.728,E2 -7221.728} C_VEL
LIN {X 0,Y 474.665,Z 341.983,A -85,B 0,C 180,E1 -7224.492,E2 -7224.492} C_VEL
LIN {X 0,Y 474.685,Z 341.983,A -85,B 0,C 180,E1 -7227.334,E2 -7227.334} C_VEL
LIN {X 0,Y 474.61,Z 341.992,A -85,B 0,C 180,E1 -7230.23,E2 -7230.23} C_VEL
LIN {X 0,Y 474.647,Z 341.988,A -85,B 0,C 180,E1 -7233.22,E2 -7233.22} C_VEL
LIN {X 0,Y 474.597,Z 341.993,A -85,B 0,C 180,E1 -7236.323,E2 -7236.323} C_VEL
LIN {X 0,Y 474.63,Z 341.986,A -85,B 0,C 180,E1 -7239.647,E2 -7239.647} C_VEL
LIN {X 0,Y 474.617,Z 341.993,A -85,B 0,C 180,E1 -7242.934,E2 -7242.934} C_VEL
LIN {X 0,Y 474.615,Z 341.995,A -85,B 0,C 180,E1 -7245.895,E2 -7245.895} C_VEL
LIN {X 0,Y 474.635,Z 341.992,A -85,B 0,C 180,E1 -7249.04,E2 -7249.04} C_VEL
LIN {X 0,Y 474.668,Z 342.207,A -85,B 0,C 180,E1 -7249.347,E2 -7249.347} C_VEL
LIN {X 0,Y 476.057,Z 349.3,A -85,B 0,C 180,E1 -7252.217,E2 -7252.217} C_VEL
LIN {X 0,Y 476.93,Z 354.323,A -85,B 0,C 180,E1 -7254.142,E2 -7254.142} C_VEL
LIN {X 0,Y 476.9,Z 359.4,A -85,B 0,C 180,E1 -7255.944,E2 -7255.944} C_VEL
LIN {X 0,Y 476.318,Z 368.177,A -85,B 0,C 180,E1 -7258.907,E2 -7258.907} C_VEL
LIN {X 0,Y 475.853,Z 377.053,A -85,B 0,C 180,E1 -7261.795,E2 -7261.795} C_VEL
LIN {X 0,Y 475.341,Z 387.402,A -85,B 0,C 180,E1 -7265.078,E2 -7265.078} C_VEL
LIN {X 0,Y 474.963,Z 396.166,A -85,B 0,C 180,E1 -7267.832,E2 -7267.832} C_VEL
LIN {X 0,Y 474.876,Z 399.115,A -85,B 0,C 180,E1 -7268.762,E2 -7268.762} C_VEL
LIN {X 0,Y 478.472,Z 415.98,A -85,B 0,C 180,E1 -7269.272,E2 -7269.272} C_VEL
LIN {X 0,Y 479.908,Z 423.449,A -85,B 0,C 180,E1 -7269.553,E2 -7269.553} C_VEL
LIN {X 0,Y 479.335,Z 438.34,A -85,B 0,C 180,E1 -7270.107,E2 -7270.107} C_VEL
LIN {X 0,Y 478.652,Z 452.81,A -85,B 0,C 180,E1 -7270.82,E2 -7270.82} C_VEL
LIN {X 0,Y 477.89,Z 466.583,A -85,B 0,C 180,E1 -7271.678,E2 -7271.678} C_VEL
LIN {X 0,Y 477.152,Z 479.279,A -85,B 0,C 180,E1 -7272.646,E2 -7272.646} C_VEL
LIN {X 0,Y 476.393,Z 492.189,A -85,B 0,C 180,E1 -7273.832,E2 -7273.832} C_VEL
LIN {X 0,Y 475.729,Z 503.024,A -85,B 0,C 180,E1 -7275.017,E2 -7275.017} C_VEL
LIN {X 0,Y 475.194,Z 513.07,A -85,B 0,C 180,E1 -7276.312,E2 -7276.312} C_VEL
LIN {X 0,Y 474.673,Z 522.443,A -85,B 0,C 180,E1 -7277.74,E2 -7277.74} C_VEL
LIN {X 0,Y 474.377,Z 531.12,A -85,B 0,C 180,E1 -7279.328,E2 -7279.328} C_VEL
LIN {X 0,Y 474.042,Z 538.765,A -85,B 0,C 180,E1 -7281.044,E2 -7281.044} C_VEL
LIN {X 0,Y 473.907,Z 544.838,A -85,B 0,C 180,E1 -7282.758,E2 -7282.758} C_VEL
LIN {X 0,Y 473.811,Z 548.431,A -85,B 0,C 180,E1 -7284.04,E2 -7284.04} C_VEL
LIN {X 0,Y 473.711,Z 552.079,A -85,B 0,C 180,E1 -7285.746,E2 -7285.746} C_VEL
LIN {X 0,Y 473.797,Z 553.438,A -85,B 0,C 180,E1 -7286.598,E2 -7286.598} C_VEL
LIN {X 0,Y 473.748,Z 555.237,A -85,B 0,C 180,E1 -7288.3,E2 -7288.3} C_VEL
LIN {X 0,Y 473.666,Z 555.848,A -85,B 0,C 180,E1 -7290,E2 -7290} C_VEL
LIN {X 0,Y 473.748,Z 555.236,A -85,B 0,C 180,E1 -7291.7,E2 -7291.7} C_VEL
LIN {X 0,Y 473.797,Z 553.439,A -85,B 0,C 180,E1 -7293.401,E2 -7293.401} C_VEL
LIN {X 0,Y 473.79,Z 550.423,A -85,B 0,C 180,E1 -7295.106,E2 -7295.106} C_VEL
LIN {X 0,Y 473.894,Z 546.127,A -85,B 0,C 180,E1 -7296.814,E2 -7296.814} C_VEL
LIN {X 0,Y 473.982,Z 540.429,A -85,B 0,C 180,E1 -7298.527,E2 -7298.527} C_VEL
LIN {X 0,Y 474.258,Z 533.187,A -85,B 0,C 180,E1 -7300.243,E2 -7300.243} C_VEL
LIN {X 0,Y 474.611,Z 525.437,A -85,B 0,C 180,E1 -7301.748,E2 -7301.748} C_VEL
LIN {X 0,Y 475.05,Z 516.108,A -85,B 0,C 180,E1 -7303.256,E2 -7303.256} C_VEL
LIN {X 0,Y 475.533,Z 506.594,A -85,B 0,C 180,E1 -7304.551,E2 -7304.551} C_VEL
LIN {X 0,Y 476.217,Z 494.352,A -85,B 0,C 180,E1 -7305.954,E2 -7305.954} C_VEL
LIN {X 0,Y 476.985,Z 481.884,A -85,B 0,C 180,E1 -7307.139,E2 -7307.139} C_VEL
LIN {X 0,Y 477.765,Z 468.161,A -85,B 0,C 180,E1 -7308.216,E2 -7308.216} C_VEL
LIN {X 0,Y 478.491,Z 454.762,A -85,B 0,C 180,E1 -7309.075,E2 -7309.075} C_VEL
LIN {X 0,Y 479.254,Z 440.454,A -85,B 0,C 180,E1 -7309.804,E2 -7309.804} C_VEL
LIN {X 0,Y 479.862,Z 425.501,A -85,B 0,C 180,E1 -7310.384,E2 -7310.384} C_VEL
LIN {X 0,Y 479.584,Z 421.256,A -85,B 0,C 180,E1 -7310.528,E2 -7310.528} C_VEL
LIN {X 0,Y 476.286,Z 405.518,A -85,B 0,C 180,E1 -7311.058,E2 -7311.058} C_VEL
LIN {X 0,Y 474.855,Z 399.044,A -85,B 0,C 180,E1 -7311.259,E2 -7311.259} C_VEL
LIN {X 0,Y 475.235,Z 390.344,A -85,B 0,C 180,E1 -7313.997,E2 -7313.997} C_VEL
LIN {X 0,Y 475.683,Z 380.024,A -85,B 0,C 180,E1 -7317.259,E2 -7317.259} C_VEL
LIN {X 0,Y 476.14,Z 371.093,A -85,B 0,C 180,E1 -7320.123,E2 -7320.123} C_VEL
LIN {X 0,Y 476.629,Z 363.008,A -85,B 0,C 180,E1 -7322.81,E2 -7322.81} C_VEL
LIN {X 0,Y 477.064,Z 356.452,A -85,B 0,C 180,E1 -7325.068,E2 -7325.068} C_VEL
LIN {X 0,Y 476.321,Z 350.691,A -85,B 0,C 180,E1 -7327.225,E2 -7327.225} C_VEL
LIN {X 0,Y 474.912,Z 343.457,A -85,B 0,C 180,E1 -7330.126,E2 -7330.126} C_VEL
LIN {X 0,Y 474.632,Z 341.99,A -85,B 0,C 180,E1 -7330.808,E2 -7330.808} C_VEL
LIN {X 0,Y 474.602,Z 341.987,A -85,B 0,C 180,E1 -7333.481,E2 -7333.481} C_VEL
LIN {X 0,Y 474.602,Z 341.992,A -85,B 0,C 180,E1 -7336.519,E2 -7336.519} C_VEL
LIN {X 0,Y 474.64,Z 341.983,A -85,B 0,C 180,E1 -7339.345,E2 -7339.345} C_VEL
LIN {X 0,Y 474.622,Z 341.991,A -85,B 0,C 180,E1 -7341.703,E2 -7341.703} C_VEL
LIN {X 0,Y 474.633,Z 341.993,A -85,B 0,C 180,E1 -7344.727,E2 -7344.727} C_VEL
LIN {X 0,Y 474.638,Z 341.993,A -85,B 0,C 180,E1 -7347.788,E2 -7347.788} C_VEL
LIN {X 0,Y 474.627,Z 341.989,A -85,B 0,C 180,E1 -7350.885,E2 -7350.885} C_VEL
LIN {X 0,Y 474.664,Z 341.983,A -85,B 0,C 180,E1 -7353.629,E2 -7353.629} C_VEL
LIN {X 0,Y 474.64,Z 341.988,A -85,B 0,C 180,E1 -7356.641,E2 -7356.641} C_VEL
LIN {X 0,Y 474.658,Z 341.984,A -85,B 0,C 180,E1 -7360.09,E2 -7360.09} C_VEL
LIN {X 0,Y 474.652,Z 341.985,A -85,B 0,C 180,E1 -7362.775,E2 -7362.775} C_VEL
LIN {X 0,Y 474.653,Z 341.983,A -85,B 0,C 180,E1 -7365.421,E2 -7365.421} C_VEL
LIN {X 0,Y 474.744,Z 341.974,A -85,B 0,C 180,E1 -7368.039,E2 -7368.039} C_VEL
LIN {X 0,Y 474.716,Z 341.98,A -85,B 0,C 180,E1 -7371.486,E2 -7371.486} C_VEL
LIN {X 0,Y 474.783,Z 341.965,A -85,B 0,C 180,E1 -7374.053,E2 -7374.053} C_VEL
LIN {X 0,Y 474.898,Z 341.95,A -85,B 0,C 180,E1 -7377.456,E2 -7377.456} C_VEL
LIN {X 0,Y 474.917,Z 341.952,A -85,B 0,C 180,E1 -7380,E2 -7380} C_VEL
LIN {X 0,Y 474.898,Z 341.953,A -85,B 0,C 180,E1 -7382.545,E2 -7382.545} C_VEL
LIN {X 0,Y 474.784,Z 341.967,A -85,B 0,C 180,E1 -7385.948,E2 -7385.948} C_VEL
LIN {X 0,Y 474.731,Z 341.977,A -85,B 0,C 180,E1 -7388.514,E2 -7388.514} C_VEL
LIN {X 0,Y 474.745,Z 341.974,A -85,B 0,C 180,E1 -7391.962,E2 -7391.962} C_VEL
LIN {X 0,Y 474.686,Z 341.979,A -85,B 0,C 180,E1 -7395.768,E2 -7395.768} C_VEL
LIN {X 0,Y 474.669,Z 341.982,A -85,B 0,C 180,E1 -7399.01,E2 -7399.01} C_VEL
LIN {X 0,Y 474.594,Z 341.993,A -85,B 0,C 180,E1 -7401.729,E2 -7401.729} C_VEL
LIN {X 0,Y 474.664,Z 341.98,A -85,B 0,C 180,E1 -7404.493,E2 -7404.493} C_VEL
LIN {X 0,Y 474.685,Z 341.98,A -85,B 0,C 180,E1 -7407.334,E2 -7407.334} C_VEL
LIN {X 0,Y 474.61,Z 341.993,A -85,B 0,C 180,E1 -7410.23,E2 -7410.23} C_VEL
LIN {X 0,Y 474.647,Z 341.987,A -85,B 0,C 180,E1 -7413.22,E2 -7413.22} C_VEL
LIN {X 0,Y 474.592,Z 341.992,A -85,B 0,C 180,E1 -7416.323,E2 -7416.323} C_VEL
LIN {X 0,Y 474.631,Z 341.988,A -85,B 0,C 180,E1 -7419.648,E2 -7419.648} C_VEL
LIN {X 0,Y 474.618,Z 341.989,A -85,B 0,C 180,E1 -7422.934,E2 -7422.934} C_VEL
LIN {X 0,Y 474.613,Z 341.992,A -85,B 0,C 180,E1 -7425.895,E2 -7425.895} C_VEL
LIN {X 0,Y 474.642,Z 341.989,A -85,B 0,C 180,E1 -7429.039,E2 -7429.039} C_VEL
LIN {X 0,Y 474.683,Z 342.169,A -85,B 0,C 180,E1 -7429.609,E2 -7429.609} C_VEL
LIN {X 0,Y 475.006,Z 345.284,A -85,B 0,C 180,E1 -7431.644,E2 -7431.644} C_VEL
LIN {X 0,Y 474.896,Z 350.169,A -85,B 0,C 180,E1 -7434.749,E2 -7434.749} C_VEL
LIN {X 0,Y 474.717,Z 355.093,A -85,B 0,C 180,E1 -7437.794,E2 -7437.794} C_VEL
LIN {X 0,Y 474.518,Z 360.262,A -85,B 0,C 180,E1 -7440.908,E2 -7440.908} C_VEL
LIN {X 0,Y 474.414,Z 364.807,A -85,B 0,C 180,E1 -7443.614,E2 -7443.614} C_VEL
LIN {X 0,Y 474.274,Z 370.237,A -85,B 0,C 180,E1 -7446.743,E2 -7446.743} C_VEL
LIN {X 0,Y 474.1,Z 376.246,A -85,B 0,C 180,E1 -7450.065,E2 -7450.065} C_VEL
LIN {X 0,Y 474.093,Z 378.199,A -85,B 0,C 180,E1 -7451.114,E2 -7451.114} C_VEL
LIN {X 0,Y 474.851,Z 379.08,A -85,B 0,C 180,E1 -7451.384,E2 -7451.384} C_VEL
LIN {X 0,Y 477.071,Z 380.868,A -85,B 0,C 180,E1 -7451.637,E2 -7451.637} C_VEL
LIN {X 0,Y 480.002,Z 383.938,A -85,B 0,C 180,E1 -7451.83,E2 -7451.83} C_VEL
LIN {X 0,Y 481.015,Z 386.707,A -85,B 0,C 180,E1 -7451.937,E2 -7451.937} C_VEL
LIN {X 0,Y 481.024,Z 387.14,A -85,B 0,C 180,E1 -7451.947,E2 -7451.947} C_VEL
LIN {X 0,Y 473.357,Z 400.914,A -85,B 0,C 180,E1 -7452.012,E2 -7452.012} C_VEL
LIN {X 0,Y 472.523,Z 406.606,A -85,B 0,C 180,E1 -7452.192,E2 -7452.192} C_VEL
LIN {X 0,Y 472.364,Z 408.56,A -85,B 0,C 180,E1 -7452.274,E2 -7452.274} C_VEL
LIN {X 0,Y 471.792,Z 421.46,A -85,B 0,C 180,E1 -7452.89,E2 -7452.89} C_VEL
LIN {X 0,Y 471.227,Z 433.747,A -85,B 0,C 180,E1 -7453.65,E2 -7453.65} C_VEL
LIN {X 0,Y 470.442,Z 446.361,A -85,B 0,C 180,E1 -7454.623,E2 -7454.623} C_VEL
LIN {X 0,Y 469.746,Z 457.68,A -85,B 0,C 180,E1 -7455.708,E2 -7455.708} C_VEL
LIN {X 0,Y 469.06,Z 467.76,A -85,B 0,C 180,E1 -7456.883,E2 -7456.883} C_VEL
LIN {X 0,Y 468.423,Z 477.798,A -85,B 0,C 180,E1 -7458.314,E2 -7458.314} C_VEL
LIN {X 0,Y 467.887,Z 485.328,A -85,B 0,C 180,E1 -7459.616,E2 -7459.616} C_VEL
LIN {X 0,Y 467.512,Z 491.555,A -85,B 0,C 180,E1 -7460.918,E2 -7460.918} C_VEL
LIN {X 0,Y 467.201,Z 496.708,A -85,B 0,C 180,E1 -7462.219,E2 -7462.219} C_VEL
LIN {X 0,Y 467.011,Z 502.129,A -85,B 0,C 180,E1 -7463.953,E2 -7463.953} C_VEL
LIN {X 0,Y 466.842,Z 506.054,A -85,B 0,C 180,E1 -7465.683,E2 -7465.683} C_VEL
LIN {X 0,Y 466.747,Z 508.614,A -85,B 0,C 180,E1 -7467.411,E2 -7467.411} C_VEL
LIN {X 0,Y 466.618,Z 509.896,A -85,B 0,C 180,E1 -7469.137,E2 -7469.137} C_VEL
LIN {X 0,Y 466.618,Z 509.932,A -85,B 0,C 180,E1 -7470.863,E2 -7470.863} C_VEL
LIN {X 0,Y 466.746,Z 508.724,A -85,B 0,C 180,E1 -7472.589,E2 -7472.589} C_VEL
LIN {X 0,Y 466.842,Z 506.235,A -85,B 0,C 180,E1 -7474.317,E2 -7474.317} C_VEL
LIN {X 0,Y 467.009,Z 502.374,A -85,B 0,C 180,E1 -7476.047,E2 -7476.047} C_VEL
LIN {X 0,Y 467.192,Z 497.031,A -85,B 0,C 180,E1 -7477.781,E2 -7477.781} C_VEL
LIN {X 0,Y 467.496,Z 491.966,A -85,B 0,C 180,E1 -7479.082,E2 -7479.082} C_VEL
LIN {X 0,Y 467.956,Z 484.637,A -85,B 0,C 180,E1 -7480.602,E2 -7480.602} C_VEL
LIN {X 0,Y 468.483,Z 476.995,A -85,B 0,C 180,E1 -7481.904,E2 -7481.904} C_VEL
LIN {X 0,Y 469.096,Z 467.271,A -85,B 0,C 180,E1 -7483.268,E2 -7483.268} C_VEL
LIN {X 0,Y 469.83,Z 456.42,A -85,B 0,C 180,E1 -7484.511,E2 -7484.511} C_VEL
LIN {X 0,Y 470.521,Z 444.827,A -85,B 0,C 180,E1 -7485.597,E2 -7485.597} C_VEL
LIN {X 0,Y 471.227,Z 433.457,A -85,B 0,C 180,E1 -7486.462,E2 -7486.462} C_VEL
LIN {X 0,Y 471.862,Z 420.079,A -85,B 0,C 180,E1 -7487.275,E2 -7487.275} C_VEL
LIN {X 0,Y 472.393,Z 406.331,A -85,B 0,C 180,E1 -7487.91,E2 -7487.91} C_VEL
LIN {X 0,Y 472.422,Z 399.347,A -85,B 0,C 180,E1 -7488.171,E2 -7488.171} C_VEL
LIN {X 0,Y 468.642,Z 384.814,A -85,B 0,C 180,E1 -7488.743,E2 -7488.743} C_VEL
LIN {X 0,Y 467.025,Z 379.003,A -85,B 0,C 180,E1 -7488.942,E2 -7488.942} C_VEL
LIN {X 0,Y 467.132,Z 373.293,A -85,B 0,C 180,E1 -7492.094,E2 -7492.094} C_VEL
LIN {X 0,Y 467.261,Z 368.356,A -85,B 0,C 180,E1 -7494.907,E2 -7494.907} C_VEL
LIN {X 0,Y 467.414,Z 363.516,A -85,B 0,C 180,E1 -7497.783,E2 -7497.783} C_VEL
LIN {X 0,Y 467.593,Z 358.126,A -85,B 0,C 180,E1 -7501.049,E2 -7501.049} C_VEL
LIN {X 0,Y 467.787,Z 352.904,A -85,B 0,C 180,E1 -7504.277,E2 -7504.277} C_VEL
LIN {X 0,Y 467.992,Z 348.196,A -85,B 0,C 180,E1 -7507.257,E2 -7507.257} C_VEL
LIN {X 0,Y 467.915,Z 345.362,A -85,B 0,C 180,E1 -7509.112,E2 -7509.112} C_VEL
LIN {X 0,Y 467.609,Z 342.87,A -85,B 0,C 180,E1 -7510.828,E2 -7510.828} C_VEL
LIN {X 0,Y 467.559,Z 342.869,A -85,B 0,C 180,E1 -7513.821,E2 -7513.821} C_VEL
LIN {X 0,Y 467.56,Z 342.87,A -85,B 0,C 180,E1 -7516.256,E2 -7516.256} C_VEL
LIN {X 0,Y 467.582,Z 342.863,A -85,B 0,C 180,E1 -7518.723,E2 -7518.723} C_VEL
LIN {X 0,Y 467.57,Z 342.866,A -85,B 0,C 180,E1 -7521.956,E2 -7521.956} C_VEL
LIN {X 0,Y 467.569,Z 342.868,A -85,B 0,C 180,E1 -7525.168,E2 -7525.168} C_VEL
LIN {X 0,Y 467.588,Z 342.868,A -85,B 0,C 180,E1 -7528.26,E2 -7528.26} C_VEL
LIN {X 0,Y 467.582,Z 342.867,A -85,B 0,C 180,E1 -7531.251,E2 -7531.251} C_VEL
LIN {X 0,Y 467.616,Z 342.859,A -85,B 0,C 180,E1 -7534.16,E2 -7534.16} C_VEL
LIN {X 0,Y 467.582,Z 342.866,A -85,B 0,C 180,E1 -7536.996,E2 -7536.996} C_VEL
LIN {X 0,Y 467.628,Z 342.859,A -85,B 0,C 180,E1 -7539.777,E2 -7539.777} C_VEL
LIN {X 0,Y 467.605,Z 342.86,A -85,B 0,C 180,E1 -7542.506,E2 -7542.506} C_VEL
LIN {X 0,Y 467.612,Z 342.863,A -85,B 0,C 180,E1 -7545.196,E2 -7545.196} C_VEL
LIN {X 0,Y 467.662,Z 342.854,A -85,B 0,C 180,E1 -7547.855,E2 -7547.855} C_VEL
LIN {X 0,Y 467.686,Z 342.852,A -85,B 0,C 180,E1 -7551.357,E2 -7551.357} C_VEL
LIN {X 0,Y 467.75,Z 342.843,A -85,B 0,C 180,E1 -7553.963,E2 -7553.963} C_VEL
LIN {X 0,Y 467.864,Z 342.828,A -85,B 0,C 180,E1 -7557.417,E2 -7557.417} C_VEL
LIN {X 0,Y 467.888,Z 342.83,A -85,B 0,C 180,E1 -7560,E2 -7560} C_VEL
LIN {X 0,Y 467.865,Z 342.829,A -85,B 0,C 180,E1 -7562.583,E2 -7562.583} C_VEL
LIN {X 0,Y 467.741,Z 342.845,A -85,B 0,C 180,E1 -7566.037,E2 -7566.037} C_VEL
LIN {X 0,Y 467.675,Z 342.857,A -85,B 0,C 180,E1 -7568.643,E2 -7568.643} C_VEL
LIN {X 0,Y 467.688,Z 342.856,A -85,B 0,C 180,E1 -7572.144,E2 -7572.144} C_VEL
LIN {X 0,Y 467.655,Z 342.858,A -85,B 0,C 180,E1 -7575.885,E2 -7575.885} C_VEL
LIN {X 0,Y 467.628,Z 342.86,A -85,B 0,C 180,E1 -7579.307,E2 -7579.307} C_VEL
LIN {X 0,Y 467.542,Z 342.873,A -85,B 0,C 180,E1 -7582.073,E2 -7582.073} C_VEL
LIN {X 0,Y 467.609,Z 342.863,A -85,B 0,C 180,E1 -7584.887,E2 -7584.887} C_VEL
LIN {X 0,Y 467.624,Z 342.86,A -85,B 0,C 180,E1 -7587.769,E2 -7587.769} C_VEL
LIN {X 0,Y 467.572,Z 342.868,A -85,B 0,C 180,E1 -7591.045,E2 -7591.045} C_VEL
LIN {X 0,Y 467.594,Z 342.866,A -85,B 0,C 180,E1 -7594.242,E2 -7594.242} C_VEL
LIN {X 0,Y 467.554,Z 342.874,A -85,B 0,C 180,E1 -7597.186,E2 -7597.186} C_VEL
LIN {X 0,Y 467.58,Z 342.868,A -85,B 0,C 180,E1 -7600.264,E2 -7600.264} C_VEL
LIN {X 0,Y 467.589,Z 342.869,A -85,B 0,C 180,E1 -7602.567,E2 -7602.567} C_VEL
LIN {X 0,Y 467.569,Z 342.866,A -85,B 0,C 180,E1 -7605.052,E2 -7605.052} C_VEL
LIN {X 0,Y 467.591,Z 342.867,A -85,B 0,C 180,E1 -7607.44,E2 -7607.44} C_VEL
LIN {X 0,Y 467.606,Z 342.927,A -85,B 0,C 180,E1 -7608.887,E2 -7608.887} C_VEL
LIN {X 0,Y 468.923,Z 349.636,A -85,B 0,C 180,E1 -7611.675,E2 -7611.675} C_VEL
LIN {X 0,Y 469.94,Z 355.181,A -85,B 0,C 180,E1 -7613.86,E2 -7613.86} C_VEL
LIN {X 0,Y 470.062,Z 359.336,A -85,B 0,C 180,E1 -7615.378,E2 -7615.378} C_VEL
LIN {X 0,Y 469.439,Z 368.593,A -85,B 0,C 180,E1 -7618.578,E2 -7618.578} C_VEL
